C01780=1012.126,212.410,-136.881,-33.428,76.064,-33.422
C01781=1012.128,212.654,-136.908,-33.436,76.075,-33.431
C01782=1012.129,212.897,-136.935,-33.444,76.085,-33.440
C01783=1012.131,213.142,-136.961,-33.452,76.095,-33.450
C01784=1012.133,213.385,-136.987,-33.459,76.106,-33.457
C01785=1012.135,213.629,-137.015,-33.468,76.116,-33.467
C01786=1012.138,213.873,-137.042,-33.476,76.127,-33.476
C01787=1012.140,214.117,-137.068,-33.485,76.137,-33.487
C01788=1012.142,214.361,-137.095,-33.493,76.147,-33.496
C01789=1012.144,214.607,-137.122,-33.501,76.158,-33.504
C01790=1012.146,214.852,-137.149,-33.509,76.168,-33.515
C01791=1012.149,215.097,-137.177,-33.518,76.179,-33.524
C01792=1012.151,215.342,-137.204,-33.526,76.189,-33.534
C01793=1012.152,215.587,-137.231,-33.534,76.200,-33.543
C01794=1012.155,215.832,-137.258,-33.543,76.210,-33.554
C01795=1012.157,216.079,-137.285,-33.552,76.221,-33.563
C01796=1012.160,216.324,-137.312,-33.561,76.231,-33.574
C01797=1012.161,216.570,-137.339,-33.569,76.242,-33.583
C01798=1012.164,216.818,-137.366,-33.577,76.253,-33.592
C01799=1012.167,217.073,-137.394,-33.584,76.263,-33.599
C01800=1012.169,217.333,-137.423,-33.593,76.274,-33.610
C01801=1012.171,217.597,-137.452,-33.601,76.285,-33.619
C01802=1012.174,217.878,-137.484,-33.611,76.297,-33.630
C01803=1012.176,218.167,-137.515,-33.622,76.309,-33.643
C01804=1012.179,218.460,-137.547,-33.633,76.322,-33.656
C01805=1012.182,218.757,-137.580,-33.644,76.334,-33.669
C01806=1012.185,219.060,-137.614,-33.655,76.346,-33.682
C01807=1012.187,219.356,-137.647,-33.666,76.358,-33.695
C01808=1012.190,219.638,-137.678,-33.676,76.370,-33.706
C01809=1012.193,219.909,-137.708,-33.686,76.382,-33.717
C01810=1012.195,220.170,-137.737,-33.693,76.393,-33.725
C01811=1012.197,220.419,-137.765,-33.702,76.404,-33.734
C01812=1012.200,220.665,-137.792,-33.709,76.414,-33.743
C01813=1012.202,220.911,-137.819,-33.718,76.424,-33.752
C01814=1012.205,221.156,-137.846,-33.727,76.434,-33.763
C01815=1012.208,221.402,-137.874,-33.736,76.444,-33.774
C01816=1012.210,221.648,-137.901,-33.743,76.454,-33.782
C01817=1012.211,221.894,-137.929,-33.753,76.464,-33.793
C01818=1012.214,222.140,-137.956,-33.761,76.474,-33.802
C01819=1012.216,222.385,-137.983,-33.769,76.483,-33.811
C01820=1012.219,222.630,-138.011,-33.778,76.493,-33.822
C01821=1012.222,222.876,-138.038,-33.785,76.503,-33.829
C01822=1012.224,223.122,-138.065,-33.794,76.513,-33.840
C01823=1012.227,223.368,-138.093,-33.803,76.524,-33.850
C01824=1012.229,223.614,-138.120,-33.812,76.534,-33.861
C01825=1012.231,223.859,-138.147,-33.822,76.545,-33.873
C01826=1012.234,224.105,-138.175,-33.831,76.556,-33.882
C01827=1012.236,224.351,-138.203,-33.840,76.566,-33.893
C01828=1012.238,224.597,-138.230,-33.849,76.575,-33.902
C01829=1012.241,224.842,-138.258,-33.857,76.585,-33.912
C01830=1012.243,225.088,-138.285,-33.864,76.595,-33.919
C01831=1012.246,225.334,-138.313,-33.873,76.605,-33.930
C01832=1012.248,225.579,-138.340,-33.883,76.615,-33.942
C01833=1012.251,225.825,-138.367,-33.890,76.625,-33.949
C01834=1012.253,226.071,-138.394,-33.900,76.635,-33.961
C01835=1012.256,226.316,-138.423,-33.908,76.646,-33.970
C01836=1012.258,226.562,-138.450,-33.918,76.656,-33.982
C01837=1012.261,226.807,-138.477,-33.928,76.667,-33.993
C01838=1012.264,227.053,-138.505,-33.937,76.677,-34.003
C01839=1012.266,227.299,-138.532,-33.945,76.686,-34.012
C01840=1012.268,227.545,-138.560,-33.953,76.695,-34.021
C01841=1012.271,227.790,-138.588,-33.962,76.706,-34.031
C01842=1012.273,228.036,-138.615,-33.970,76.715,-34.041
C01843=1012.276,228.282,-138.642,-33.980,76.725,-34.052
C01844=1012.279,228.527,-138.671,-33.990,76.735,-34.064
C01845=1012.281,228.773,-138.698,-33.998,76.746,-34.073
C01846=1012.284,229.018,-138.726,-34.007,76.757,-34.083
C01847=1012.286,229.264,-138.753,-34.017,76.767,-34.095
C01848=1012.289,229.510,-138.780,-34.026,76.777,-34.105
C01849=1012.291,229.755,-138.808,-34.034,76.787,-34.114
C01850=1012.294,230.001,-138.836,-34.043,76.796,-34.124
C01851=1012.297,230.246,-138.863,-34.051,76.805,-34.133
C01852=1012.300,230.492,-138.891,-34.061,76.815,-34.145
C01853=1012.301,230.738,-138.919,-34.069,76.824,-34.154
C01854=1012.304,230.984,-138.947,-34.079,76.834,-34.166
C01855=1012.307,231.229,-138.974,-34.087,76.844,-34.174
C01856=1012.310,231.475,-139.002,-34.097,76.854,-34.186
C01857=1012.313,231.721,-139.030,-34.106,76.865,-34.196
C01858=1012.315,231.966,-139.057,-34.116,76.875,-34.208
C01859=1012.318,232.212,-139.085,-34.125,76.886,-34.218
C01860=1012.320,232.457,-139.113,-34.134,76.895,-34.227
C01861=1012.323,232.703,-139.141,-34.142,76.904,-34.237
C01862=1012.326,232.948,-139.168,-34.152,76.913,-34.248
C01863=1012.329,233.193,-139.197,-34.161,76.924,-34.259
C01864=1012.332,233.439,-139.224,-34.169,76.933,-34.268
C01865=1012.334,233.684,-139.252,-34.179,76.943,-34.280
C01866=1012.337,233.931,-139.279,-34.188,76.952,-34.290
C01867=1012.340,234.175,-139.307,-34.197,76.963,-34.300
C01868=1012.342,234.421,-139.336,-34.207,76.973,-34.312
C01869=1012.345,234.668,-139.363,-34.217,76.983,-34.322
C01870=1012.347,234.912,-139.391,-34.227,76.993,-34.334
C01871=1012.350,235.158,-139.419,-34.236,77.003,-34.344
C01872=1012.353,235.404,-139.447,-34.244,77.012,-34.354
C01873=1012.356,235.649,-139.475,-34.253,77.021,-34.364
C01874=1012.359,235.895,-139.503,-34.262,77.030,-34.374
C01875=1012.361,236.140,-139.531,-34.270,77.039,-34.384
C01876=1012.364,236.385,-139.559,-34.281,77.049,-34.396
C01877=1012.368,236.631,-139.587,-34.290,77.060,-34.406
C01878=1012.370,236.876,-139.614,-34.299,77.069,-34.416
C01879=1012.373,237.122,-139.642,-34.308,77.080,-34.426
C01880=1012.376,237.368,-139.670,-34.320,77.091,-34.441
C01881=1012.378,237.612,-139.698,-34.328,77.099,-34.449
C01882=1012.382,237.858,-139.726,-34.336,77.109,-34.459
C01883=1012.385,238.104,-139.754,-34.345,77.118,-34.469
C01884=1012.387,238.350,-139.782,-34.355,77.126,-34.481
C01885=1012.389,238.595,-139.810,-34.364,77.135,-34.491
C01886=1012.392,238.841,-139.838,-34.373,77.146,-34.501
C01887=1012.396,239.086,-139.867,-34.382,77.155,-34.511
C01888=1012.398,239.331,-139.894,-34.393,77.165,-34.524
C01889=1012.401,239.577,-139.923,-34.403,77.176,-34.534
C01890=1012.404,239.822,-139.951,-34.413,77.186,-34.546
C01891=1012.407,240.067,-139.979,-34.423,77.197,-34.557
C01892=1012.410,240.313,-140.007,-34.431,77.204,-34.567
C01893=1012.413,240.558,-140.035,-34.440,77.213,-34.577
C01894=1012.416,240.804,-140.063,-34.449,77.223,-34.587
C01895=1012.419,241.050,-140.091,-34.458,77.232,-34.598
C01896=1012.422,241.295,-140.119,-34.467,77.241,-34.608
C01897=1012.425,241.540,-140.147,-34.478,77.251,-34.620
C01898=1012.428,241.786,-140.175,-34.487,77.260,-34.631
C01899=1012.431,242.031,-140.204,-34.498,77.270,-34.643
C01900=1012.434,242.276,-140.231,-34.507,77.281,-34.654
C01901=1012.436,242.522,-140.260,-34.518,77.291,-34.666
C01902=1012.439,242.768,-140.288,-34.526,77.301,-34.675
C01903=1012.443,243.013,-140.317,-34.536,77.309,-34.687
C01904=1012.446,243.258,-140.345,-34.544,77.318,-34.695
C01905=1012.448,243.503,-140.373,-34.554,77.326,-34.708
C01906=1012.451,243.749,-140.401,-34.563,77.335,-34.718
C01907=1012.454,243.994,-140.429,-34.573,77.344,-34.728
C01908=1012.457,244.240,-140.458,-34.583,77.354,-34.741
C01909=1012.461,244.485,-140.486,-34.592,77.364,-34.750
C01910=1012.464,244.731,-140.515,-34.603,77.374,-34.762
C01911=1012.467,244.975,-140.542,-34.614,77.384,-34.775
C01912=1012.470,245.221,-140.571,-34.624,77.395,-34.786
C01913=1012.473,245.466,-140.600,-34.633,77.404,-34.797
C01914=1012.476,245.712,-140.628,-34.641,77.412,-34.807
C01915=1012.479,245.957,-140.656,-34.651,77.421,-34.817
C01916=1012.482,246.203,-140.685,-34.659,77.429,-34.826
C01917=1012.485,246.448,-140.714,-34.668,77.438,-34.836
C01918=1012.488,246.694,-140.742,-34.678,77.447,-34.849
C01919=1012.491,246.939,-140.769,-34.688,77.457,-34.860
C01920=1012.494,247.184,-140.798,-34.698,77.467,-34.871
C01921=1012.497,247.429,-140.827,-34.709,77.477,-34.884
C01922=1012.500,247.675,-140.855,-34.719,77.487,-34.895
C01923=1012.504,247.920,-140.884,-34.730,77.497,-34.908
C01924=1012.507,248.165,-140.912,-34.738,77.506,-34.916
C01925=1012.510,248.410,-140.941,-34.749,77.514,-34.929
C01926=1012.513,248.656,-140.969,-34.756,77.522,-34.937
C01927=1012.517,248.901,-140.998,-34.767,77.531,-34.950
C01928=1012.520,249.147,-141.026,-34.776,77.540,-34.961
C01929=1012.523,249.391,-141.055,-34.786,77.549,-34.971
C01930=1012.526,249.637,-141.083,-34.796,77.558,-34.982
C01931=1012.529,249.883,-141.112,-34.807,77.568,-34.995
C01932=1012.532,250.128,-141.141,-34.817,77.579,-35.007
C01933=1012.535,250.374,-141.169,-34.827,77.588,-35.017
C01934=1012.539,250.619,-141.198,-34.838,77.598,-35.031
C01935=1012.542,250.864,-141.226,-34.846,77.606,-35.039
C01936=1012.545,251.109,-141.255,-34.857,77.615,-35.052
C01937=1012.549,251.354,-141.284,-34.865,77.623,-35.061
C01938=1012.552,251.600,-141.312,-34.875,77.631,-35.073
C01939=1012.555,251.845,-141.341,-34.885,77.640,-35.084
C01940=1012.559,252.090,-141.369,-34.895,77.650,-35.095
C01941=1012.562,252.335,-141.398,-34.905,77.659,-35.106
C01942=1012.565,252.580,-141.427,-34.916,77.669,-35.120
C01943=1012.568,252.826,-141.455,-34.925,77.679,-35.129
C01944=1012.571,253.071,-141.484,-34.937,77.689,-35.142
C01945=1012.575,253.316,-141.513,-34.946,77.698,-35.153
C01946=1012.578,253.562,-141.541,-34.956,77.705,-35.164
C01947=1012.581,253.807,-141.570,-34.965,77.714,-35.175
C01948=1012.584,254.052,-141.599,-34.974,77.722,-35.186
C01949=1012.588,254.297,-141.628,-34.984,77.731,-35.197
C01950=1012.591,254.542,-141.656,-34.994,77.740,-35.208
C01951=1012.594,254.787,-141.685,-35.004,77.749,-35.219
C01952=1012.598,255.032,-141.714,-35.014,77.759,-35.231
C01953=1012.602,255.278,-141.743,-35.026,77.768,-35.244
C01954=1012.605,255.523,-141.773,-35.036,77.778,-35.255
C01955=1012.608,255.769,-141.801,-35.047,77.788,-35.267
C01956=1012.611,256.014,-141.830,-35.058,77.797,-35.280
C01957=1012.615,256.259,-141.858,-35.066,77.805,-35.289
C01958=1012.618,256.504,-141.887,-35.075,77.813,-35.300
C01959=1012.621,256.749,-141.916,-35.085,77.822,-35.311
C01960=1012.625,256.994,-141.945,-35.095,77.829,-35.322
C01961=1012.629,257.239,-141.974,-35.105,77.838,-35.334
C01962=1012.632,257.484,-142.003,-35.115,77.848,-35.345
C01963=1012.635,257.730,-142.031,-35.125,77.857,-35.356
C01964=1012.638,257.975,-142.061,-35.137,77.867,-35.370
C01965=1012.641,258.220,-142.090,-35.149,77.876,-35.384
C01966=1012.645,258.466,-142.119,-35.158,77.886,-35.393
C01967=1012.659,259.701,-142.272,-34.356,78.117,-34.079
C01968=1012.662,260.109,-142.326,-34.065,78.179,-33.616
C01969=1012.663,260.518,-142.380,-33.799,78.275,-33.178
C01970=1012.664,260.926,-142.437,-33.509,78.350,-32.716
C01971=1012.663,261.334,-142.494,-33.211,78.423,-32.244
C01972=1012.662,261.743,-142.552,-32.937,78.531,-31.799
C01973=1012.659,262.151,-142.613,-32.628,78.602,-31.316
C01974=1012.656,262.559,-142.674,-32.326,78.691,-30.842
C01975=1012.652,262.968,-142.738,-32.000,78.752,-30.341
C01976=1012.647,263.375,-142.801,-31.691,78.850,-29.859
C01977=1012.641,263.782,-142.869,-31.353,78.913,-29.346
C01978=1012.634,264.190,-142.936,-31.022,78.991,-28.841
C01979=1012.626,264.598,-143.004,-30.698,79.097,-28.344
C01980=1012.617,265.005,-143.076,-30.337,79.150,-27.807
C01981=1012.607,265.413,-143.146,-29.992,79.240,-27.288
C01982=1012.595,265.819,-143.219,-29.639,79.333,-26.761
C01983=1012.583,266.227,-143.293,-29.273,79.414,-26.220
C01984=1012.570,266.634,-143.369,-28.897,79.484,-25.668
C01985=1012.557,267.041,-143.447,-28.513,79.562,-25.107
C01986=1012.542,267.447,-143.526,-28.130,79.653,-24.550
C01987=1012.526,267.853,-143.606,-27.726,79.712,-23.968
C01988=1012.509,268.259,-143.688,-27.327,79.807,-23.393
C01989=1012.491,268.665,-143.771,-26.911,79.882,-22.800
C01990=1012.472,269.072,-143.856,-26.488,79.952,-22.199
C01991=1012.452,269.478,-143.941,-26.063,80.058,-21.600
C01992=1012.431,269.883,-144.028,-25.620,80.129,-20.978
C01993=1012.409,270.288,-144.117,-25.170,80.220,-20.351
C01994=1012.386,270.694,-144.209,-24.709,80.277,-19.709
C01995=1012.361,271.098,-144.300,-24.242,80.371,-19.066
C01996=1012.337,271.504,-144.394,-23.762,80.439,-18.406
C01997=1012.311,271.908,-144.488,-23.272,80.520,-17.736
C01998=1012.284,272.313,-144.584,-22.768,80.606,-17.054
C01999=1012.255,272.717,-144.682,-22.257,80.673,-16.361
C02000=1012.227,273.121,-144.780,-21.728,80.775,-15.656
C02001=1012.197,273.526,-144.881,-21.193,80.845,-14.939
C02002=1012.165,273.929,-144.984,-20.642,80.918,-14.206
C02003=1012.133,274.333,-145.088,-20.080,80.993,-13.462
C02004=1012.099,274.736,-145.192,-19.496,81.082,-12.698
C02005=1012.065,275.140,-145.300,-18.902,81.160,-11.919
C02006=1012.030,275.542,-145.408,-18.296,81.231,-11.129
C02007=1011.993,275.945,-145.518,-17.671,81.309,-10.319
C02008=1011.955,276.347,-145.629,-17.029,81.388,-9.493
C02009=1011.916,276.749,-145.742,-16.370,81.468,-8.648
C02010=1011.877,277.150,-145.857,-15.699,81.540,-7.791
C02011=1011.836,277.552,-145.972,-14.999,81.625,-6.906
C02012=1011.794,277.954,-146.091,-14.306,81.682,-6.021
///RCONF 0,0,0,0,0,0,0,0,0,0,0,0,0,0,0,0,0,0,0,0,0,0,0,0
C02013=1011.751,278.355,-146.209,-13.561,81.772,-5.092
C02014=1011.707,278.755,-146.330,-12.812,81.847,-4.154
C02015=1011.662,279.156,-146.453,-12.063,81.908,-3.213
C02016=1011.615,279.556,-146.576,-11.266,81.987,-2.228
C02017=1011.568,279.956,-146.702,-10.466,82.055,-1.236
C02018=1011.520,280.355,-146.828,-9.621,82.131,-0.200
C02019=1011.469,280.754,-146.957,-8.748,82.208,0.865
C02020=1011.418,281.153,-147.087,-7.854,82.282,1.952
C02021=1011.366,281.551,-147.219,-6.951,82.345,3.054
C02022=1011.313,281.949,-147.352,-5.979,82.425,4.221
C02023=1011.286,282.148,-147.420,-5.489,82.462,4.808
C02024=1011.258,282.347,-147.487,-5.001,82.493,5.398
C02025=1011.231,282.546,-147.556,-4.501,82.528,5.997
C02026=1011.202,282.744,-147.624,-3.990,82.563,6.608
C02027=1011.174,282.943,-147.693,-3.493,82.589,7.207
C02028=1011.145,283.140,-147.763,-2.965,82.625,7.834
C02029=1011.117,283.339,-147.832,-2.417,82.663,8.482
C02030=1011.088,283.536,-147.903,-1.899,82.688,9.103
C02031=1011.058,283.735,-147.974,-1.341,82.723,9.762
C02032=1011.028,283.933,-148.044,-0.760,82.763,10.442
C02033=1010.998,284.131,-148.116,-0.205,82.791,11.101
C02034=1010.968,284.328,-148.188,0.380,82.825,11.786
C02035=1010.937,284.526,-148.261,0.936,82.848,12.448
C02036=1010.906,284.724,-148.333,1.533,82.881,13.146
C02037=1010.875,284.921,-148.407,2.133,82.910,13.849
C02038=1010.843,285.118,-148.481,2.711,82.931,14.533
C02039=1010.811,285.314,-148.556,3.329,82.960,15.256
C02040=1010.779,285.512,-148.629,3.994,82.998,16.021
C02041=1010.746,285.709,-148.704,4.634,83.026,16.764
C02042=1010.713,285.905,-148.781,5.281,83.054,17.515
C02043=1010.681,286.101,-148.856,5.929,83.078,18.270
C02044=1010.646,286.298,-148.933,6.600,83.104,19.047
C02045=1010.612,286.494,-149.010,7.280,83.130,19.833
C02046=1010.579,286.690,-149.088,7.927,83.145,20.590
C02047=1010.544,286.886,-149.166,8.623,83.169,21.393
C02048=1010.508,287.083,-149.243,9.382,83.202,22.256
C02049=1010.474,287.278,-149.322,10.083,83.219,23.067
C02050=1010.438,287.473,-149.402,10.786,83.235,23.882
C02051=1010.403,287.669,-149.481,11.547,83.260,24.750
C02052=1010.366,287.864,-149.560,12.362,83.290,25.670
C02053=1010.329,288.059,-149.642,13.098,83.304,26.518
C02054=1010.292,288.254,-149.722,13.896,83.326,27.424
C02055=1010.256,288.449,-149.804,14.648,83.337,28.290
C02056=1010.218,288.644,-149.886,15.421,83.350,29.176
C02057=1010.179,288.838,-149.968,16.267,83.370,30.130
C02058=1010.141,289.032,-150.051,17.100,83.386,31.073
C02059=1010.103,289.226,-150.135,17.936,83.400,32.020
C02060=1010.064,289.420,-150.218,18.754,83.409,32.953
C02061=1010.025,289.614,-150.303,19.617,83.421,33.928
C02062=1009.985,289.808,-150.388,20.451,83.428,34.877
C02063=1009.945,290.001,-150.473,21.322,83.435,35.864
C02064=1009.905,290.195,-150.559,22.218,83.443,36.873
C02065=1009.863,290.387,-150.646,23.058,83.443,37.831
C02066=1009.822,290.580,-150.733,23.981,83.450,38.868
C02067=1009.781,290.773,-150.820,24.882,83.451,39.885
C02068=1009.739,290.965,-150.908,25.775,83.449,40.896
C02069=1009.697,291.158,-150.996,26.753,83.453,41.989
C02070=1009.654,291.350,-151.085,27.660,83.449,43.015
C02071=1009.611,291.542,-151.174,28.628,83.446,44.100
C02072=1009.568,291.733,-151.265,29.517,83.435,45.111
C02073=1009.525,291.925,-151.356,30.507,83.430,46.219
C02074=1009.480,292.117,-151.446,31.413,83.416,47.248
C02075=1009.436,292.307,-151.539,32.334,83.401,48.291
C02076=1009.391,292.498,-151.630,33.357,83.392,49.433
C02077=1009.346,292.689,-151.723,34.361,83.379,50.555
C02078=1009.300,292.879,-151.815,35.346,83.362,51.662
C02079=1009.254,293.069,-151.910,36.301,83.341,52.740
C02080=1009.208,293.259,-152.004,37.296,83.320,53.859
C02081=1009.161,293.449,-152.098,38.275,83.295,54.962
C02082=1009.114,293.639,-152.194,39.247,83.269,56.059
C02083=1009.066,293.828,-152.290,40.282,83.243,57.217
C02084=1009.018,294.017,-152.386,41.233,83.210,58.296
C02085=1008.970,294.205,-152.483,42.268,83.181,59.453
C02086=1008.921,294.394,-152.581,43.222,83.144,60.537
C02087=1008.871,294.582,-152.679,44.231,83.108,61.672
C02088=1008.822,294.770,-152.778,45.232,83.070,62.798
C02089=1008.772,294.958,-152.876,46.245,83.029,63.938
C02090=1008.721,295.145,-152.977,47.183,82.983,65.008
C02091=1008.670,295.333,-153.077,48.203,82.938,66.154
C02092=1008.619,295.519,-153.179,49.113,82.886,67.199
C02093=1008.567,295.707,-153.281,50.086,82.835,68.300
C02094=1008.515,295.893,-153.382,51.138,82.786,69.476
C02095=1008.462,296.079,-153.485,52.083,82.728,70.554
C02096=1008.409,296.265,-153.588,53.034,82.670,71.635
C02097=1008.356,296.451,-153.692,53.992,82.610,72.725
C02098=1008.302,296.635,-153.798,54.922,82.546,73.787
C02099=1008.247,296.821,-153.903,55.868,82.480,74.865
C02100=1008.193,297.006,-154.009,56.789,82.411,75.920
C02101=1008.138,297.189,-154.115,57.702,82.340,76.967
C02102=1008.082,297.374,-154.222,58.657,82.268,78.053
C02103=1008.025,297.557,-154.330,59.493,82.190,79.028
C02104=1007.969,297.741,-154.438,60.423,82.113,80.089
C02105=1007.912,297.925,-154.547,61.329,82.032,81.129
C02106=1007.855,298.107,-154.657,62.166,81.948,82.104
C02107=1007.797,298.289,-154.767,63.085,81.864,83.153
C02108=1007.738,298.471,-154.878,63.950,81.776,84.153
C02109=1007.679,298.653,-154.989,64.822,81.686,85.159
C02110=1007.620,298.835,-155.101,65.608,81.592,86.085
C02111=1007.559,299.016,-155.214,66.450,81.496,87.062
C02112=1007.499,299.196,-155.327,67.303,81.399,88.048
C02113=1007.439,299.377,-155.440,68.132,81.299,89.011
C02114=1007.377,299.558,-155.556,68.904,81.195,89.923
C02115=1007.315,299.737,-155.671,69.683,81.090,90.839
C02116=1007.253,299.917,-155.786,70.456,80.982,91.748
C02117=1007.190,300.095,-155.903,71.208,80.872,92.639
C02118=1007.128,300.274,-156.021,71.962,80.760,93.530
C02119=1007.064,300.452,-156.139,72.695,80.645,94.402
C02120=1006.999,300.630,-156.257,73.408,80.527,95.254
C02121=1006.934,300.807,-156.376,74.180,80.408,96.158
C02122=1006.870,300.984,-156.496,74.851,80.286,96.971
C02123=1006.804,301.161,-156.617,75.585,80.161,97.838
C02124=1006.738,301.337,-156.738,76.228,80.036,98.624
C02125=1006.671,301.513,-156.860,76.950,79.906,99.478
C02126=1006.604,301.689,-156.983,77.596,79.776,100.264
C02127=1006.536,301.863,-157.106,78.232,79.642,101.040
C02128=1006.468,302.038,-157.230,78.893,79.506,101.838
C02129=1006.399,302.212,-157.355,79.481,79.369,102.570
C02130=1006.330,302.387,-157.480,80.107,79.229,103.332
C02131=1006.260,302.559,-157.606,80.749,79.087,104.107
C02132=1006.190,302.733,-157.733,81.359,78.943,104.854
C02133=1006.120,302.905,-157.860,81.925,78.797,105.560
C02134=1006.048,303.076,-157.988,82.506,78.649,106.278
C02135=1005.976,303.247,-158.117,83.069,78.499,106.979
C02136=1005.904,303.418,-158.246,83.618,78.347,107.667
C02137=1005.832,303.589,-158.376,84.164,78.194,108.349
C02138=1005.758,303.759,-158.507,84.697,78.038,109.019
C02139=1005.684,303.929,-158.639,85.209,77.880,109.672
C02140=1005.610,304.098,-158.770,85.770,77.719,110.361
C02141=1005.535,304.267,-158.904,86.250,77.559,110.982
C02142=1005.460,304.434,-159.037,86.784,77.394,111.645
C02143=1005.384,304.602,-159.172,87.243,77.229,112.247
C02144=1005.307,304.769,-159.306,87.757,77.061,112.890
C02145=1005.231,304.935,-159.443,88.224,76.892,113.494
C02146=1005.152,305.101,-159.579,88.679,76.722,114.086
C02147=1005.075,305.267,-159.715,89.148,76.549,114.686
C02148=1004.996,305.431,-159.854,89.565,76.377,115.243
C02149=1004.917,305.596,-159.992,90.008,76.201,115.819
C02150=1004.837,305.759,-160.131,90.470,76.023,116.407
C02151=1004.758,305.923,-160.271,90.900,75.845,116.967
C02152=1004.677,306.086,-160.412,91.302,75.666,117.503
C02153=1004.595,306.247,-160.552,91.711,75.484,118.043
C02154=1004.513,306.409,-160.694,92.113,75.301,118.576
C02155=1004.432,306.570,-160.837,92.500,75.118,119.093
C02156=1004.349,306.730,-160.981,92.888,74.932,119.611
C02157=1004.265,306.889,-161.125,93.267,74.745,120.119
C02158=1004.182,307.049,-161.270,93.628,74.557,120.612
C02159=1004.098,307.207,-161.414,94.031,74.366,121.133
C02160=1004.013,307.365,-161.561,94.357,74.177,121.596
C02161=1003.928,307.523,-161.707,94.734,73.983,122.093
C02162=1003.842,307.679,-161.854,95.069,73.790,122.558
C02163=1003.755,307.835,-162.002,95.414,73.595,123.028
C02164=1003.668,307.990,-162.150,95.770,73.398,123.502
C02165=1003.581,308.145,-162.300,96.104,73.201,123.959
C02166=1003.493,308.299,-162.451,96.409,73.005,124.391
C02167=1003.404,308.452,-162.601,96.737,72.806,124.839
C02168=1003.315,308.605,-162.752,97.028,72.608,125.256
C02169=1003.225,308.757,-162.904,97.324,72.409,125.675
C02170=1003.136,308.909,-163.056,97.664,72.207,126.122
C02171=1002.979,309.171,-163.323,98.183,71.856,126.844
C02172=1002.819,309.430,-163.591,98.681,71.503,127.543
C02173=1003.018,309.121,-163.890,77.094,71.863,112.900
C02174=1003.161,308.887,-163.649,76.172,72.173,111.744
C02175=1003.302,308.651,-163.409,75.210,72.476,110.550
C02176=1003.392,308.501,-163.258,74.548,72.665,109.749
C02177=1003.481,308.350,-163.107,73.924,72.852,108.972
C02178=1003.569,308.198,-162.955,73.303,73.038,108.192
C02179=1003.657,308.046,-162.806,72.631,73.220,107.370
C02180=1003.745,307.893,-162.657,71.982,73.400,106.562
C02181=1003.831,307.739,-162.508,71.294,73.578,105.719
C02182=1003.918,307.585,-162.361,70.582,73.751,104.857
C02183=1004.004,307.429,-162.214,69.873,73.922,103.991
C02184=1004.090,307.274,-162.067,69.167,74.092,103.123
C02185=1004.174,307.117,-161.922,68.410,74.257,102.212
C02186=1004.258,306.960,-161.776,67.703,74.421,101.336
C02187=1004.342,306.802,-161.632,66.915,74.579,100.395
C02188=1004.425,306.645,-161.488,66.163,74.735,99.479
C02189=1004.508,306.485,-161.345,65.388,74.887,98.543
C02190=1004.590,306.327,-161.203,64.598,75.036,97.590
C02191=1004.672,306.167,-161.061,63.808,75.181,96.636
C02192=1004.753,306.006,-160.920,62.999,75.324,95.661
C02193=1004.834,305.845,-160.780,62.174,75.462,94.673
C02194=1004.914,305.683,-160.639,61.357,75.598,93.687
C02195=1004.993,305.521,-160.501,60.507,75.728,92.674
C02196=1005.073,305.358,-160.362,59.625,75.854,91.630
C02197=1005.151,305.195,-160.226,58.758,75.978,90.598
C02198=1005.229,305.031,-160.088,57.910,76.100,89.575
C02199=1005.307,304.866,-159.952,57.018,76.215,88.518
C02200=1005.384,304.701,-159.816,56.131,76.328,87.459
C02201=1005.460,304.535,-159.681,55.236,76.438,86.393
C02202=1005.536,304.370,-159.548,54.297,76.540,85.291
C02203=1005.611,304.203,-159.413,53.405,76.643,84.223
C02204=1005.687,304.036,-159.281,52.450,76.737,83.103
C02205=1005.761,303.868,-159.148,51.546,76.831,82.024
C02206=1005.835,303.700,-159.018,50.569,76.917,80.883
C02207=1005.908,303.532,-158.886,49.640,77.002,79.780
C02208=1005.981,303.363,-158.757,48.693,77.083,78.660
C02209=1006.053,303.193,-158.628,47.738,77.159,77.534
C02210=1006.125,303.024,-158.498,46.789,77.233,76.412
C02211=1006.196,302.853,-158.371,45.831,77.301,75.282
C02212=1006.267,302.682,-158.244,44.865,77.365,74.144
C02213=1006.338,302.511,-158.116,43.918,77.428,73.021
C02214=1006.407,302.339,-157.990,42.937,77.484,71.868
C02215=1006.477,302.166,-157.865,41.940,77.534,70.703
C02216=1006.545,301.994,-157.741,40.968,77.582,69.560
C02217=1006.613,301.821,-157.616,40.027,77.631,68.439
C02218=1006.681,301.647,-157.494,39.047,77.670,67.289
C02219=1006.748,301.473,-157.370,38.094,77.710,66.162
C02220=1006.815,301.298,-157.249,37.138,77.745,65.030
C02221=1006.882,301.123,-157.128,36.143,77.771,63.867
C02222=1006.947,300.948,-157.006,35.217,77.802,62.764
C02223=1007.013,300.773,-156.887,34.240,77.821,61.619
C02224=1007.077,300.597,-156.768,33.314,77.844,60.517
C02225=1007.142,300.420,-156.650,32.341,77.856,59.376
C02226=1007.205,300.244,-156.531,31.418,77.871,58.279
C02227=1007.269,300.066,-156.414,30.495,77.882,57.183
C02228=1007.332,299.888,-156.297,29.571,77.888,56.088
C02229=1007.394,299.710,-156.181,28.661,77.893,55.005
C02230=1007.456,299.532,-156.066,27.756,77.894,53.928
C02231=1007.517,299.353,-155.951,26.858,77.892,52.859
C02232=1007.578,299.174,-155.837,25.983,77.890,51.811
C02233=1007.638,298.994,-155.723,25.092,77.881,50.750
C02234=1007.698,298.815,-155.611,24.204,77.867,49.695
C02235=1007.758,298.634,-155.499,23.334,77.853,48.656
C02236=1007.817,298.454,-155.387,22.510,77.843,47.658
C02237=1007.875,298.273,-155.277,21.655,77.822,46.636
C02238=1007.934,298.091,-155.166,20.824,77.802,45.636
C02239=1007.992,297.910,-155.058,19.979,77.774,44.626
C02240=1008.048,297.728,-154.948,19.193,77.754,43.669
C02241=1008.105,297.546,-154.840,18.390,77.726,42.700
C02242=1008.162,297.363,-154.732,17.590,77.694,41.735
C02243=1008.217,297.181,-154.625,16.842,77.671,40.814
C02244=1008.272,296.998,-154.519,16.062,77.635,39.871
C02245=1008.327,296.813,-154.413,15.317,77.602,38.959
C02246=1008.382,296.631,-154.307,14.584,77.569,38.059
C02247=1008.436,296.446,-154.203,13.851,77.530,37.162
C02248=1008.489,296.262,-154.098,13.140,77.493,36.285
C02249=1008.543,296.078,-153.995,12.431,77.453,35.412
C02250=1008.596,295.892,-153.892,11.735,77.411,34.552
C02251=1008.648,295.707,-153.789,11.063,77.371,33.716
C02252=1008.700,295.522,-153.688,10.360,77.317,32.856
C02253=1008.751,295.335,-153.587,9.699,77.272,32.032
C02254=1008.803,295.150,-153.486,9.077,77.233,31.245
C02255=1008.853,294.964,-153.386,8.421,77.180,30.431
C02256=1008.903,294.776,-153.286,7.813,77.138,29.660
C02257=1008.953,294.590,-153.188,7.191,77.086,28.880
C02258=1009.002,294.402,-153.090,6.576,77.033,28.107
C02259=1009.052,294.215,-152.992,5.976,76.979,27.351
C02260=1009.100,294.027,-152.894,5.406,76.932,26.619
C02261=1009.148,293.839,-152.798,4.814,76.872,25.874
C02262=1009.196,293.652,-152.702,4.267,76.824,25.168
C02263=1009.243,293.463,-152.607,3.703,76.765,24.451
C02264=1009.290,293.275,-152.512,3.160,76.711,23.751
C02265=1009.337,293.086,-152.417,2.630,76.658,23.067
C02266=1009.383,292.897,-152.323,2.104,76.600,22.388
C02267=1009.429,292.707,-152.230,1.595,76.546,21.724
C02268=1009.474,292.518,-152.138,1.089,76.488,21.065
C02269=1009.519,292.328,-152.046,0.585,76.427,20.412
C02270=1009.564,292.137,-151.954,0.085,76.362,19.765
C02271=1009.608,291.948,-151.863,-0.381,76.309,19.146
C02272=1009.651,291.757,-151.772,-0.839,76.256,18.537
C02273=1009.695,291.567,-151.682,-1.306,76.194,17.923
C02274=1009.739,291.376,-151.592,-1.745,76.141,17.332
C02275=1009.782,291.185,-151.503,-2.198,76.078,16.733
C02276=1009.823,290.993,-151.415,-2.627,76.022,16.156
C02277=1009.866,290.802,-151.327,-3.071,75.954,15.568
C02278=1009.907,290.611,-151.239,-3.488,75.897,15.005
C02279=1009.948,290.419,-151.152,-3.897,75.839,14.450
C02280=1009.990,290.226,-151.066,-4.311,75.774,13.893
C02281=1010.030,290.034,-150.980,-4.699,75.721,13.358
C02282=1010.071,289.842,-150.894,-5.094,75.657,12.822
C02283=1010.110,289.649,-150.808,-5.476,75.598,12.298
C02284=1010.149,289.456,-150.724,-5.851,75.541,11.780
C02285=1010.189,289.263,-150.640,-6.226,75.478,11.264
C02286=1010.227,289.070,-150.557,-6.583,75.421,10.767
C02287=1010.266,288.877,-150.474,-6.943,75.360,10.266
C02288=1010.305,288.683,-150.391,-7.301,75.296,9.771
C02289=1010.341,288.489,-150.309,-7.655,75.230,9.280
C02290=1010.379,288.296,-150.227,-7.991,75.173,8.805
C02291=1010.416,288.101,-150.146,-8.317,75.120,8.339
C02292=1010.453,287.907,-150.066,-8.650,75.056,7.870
C02293=1010.489,287.713,-149.985,-8.967,75.003,7.415
C02294=1010.526,287.518,-149.906,-9.300,74.931,6.949
C02295=1010.561,287.324,-149.826,-9.618,74.867,6.498
C02296=1010.596,287.129,-149.748,-9.919,74.814,6.059
C02297=1010.632,286.934,-149.668,-10.214,74.761,5.627
C02298=1010.666,286.739,-149.591,-10.525,74.691,5.185
C02299=1010.701,286.544,-149.514,-10.816,74.633,4.763
C02300=1010.735,286.349,-149.436,-11.094,74.584,4.348
C02301=1010.768,286.153,-149.360,-11.376,74.526,3.934
C02302=1010.801,285.957,-149.283,-11.655,74.467,3.523
C02303=1010.834,285.761,-149.208,-11.927,74.413,3.120
C02304=1010.867,285.566,-149.132,-12.198,74.353,2.719
C02305=1010.900,285.369,-149.057,-12.462,74.296,2.326
C02306=1010.932,285.173,-148.984,-12.733,74.228,1.929
C02307=1010.964,284.977,-148.910,-12.991,74.170,1.542
C02308=1010.995,284.781,-148.836,-13.237,74.123,1.164
C02309=1011.027,284.584,-148.763,-13.486,74.067,0.788
C02310=1011.058,284.387,-148.690,-13.735,74.009,0.411
C02311=1011.089,284.190,-148.618,-13.972,73.960,0.045
C02312=1011.119,283.993,-148.546,-14.214,73.900,-0.323
///RCONF 0,0,0,0,1,0,0,0,0,0,0,0,0,0,0,0,0,0,0,0,0,0,0,0
C02313=1011.149,283.797,-148.474,-14.449,73.848,-0.686
C02314=1011.208,283.402,-148.334,-14.919,73.727,-1.405
C02315=1011.265,283.007,-148.194,-15.367,73.620,-2.105
C02316=1011.322,282.612,-148.056,-15.803,73.514,-2.791
C02317=1011.377,282.216,-147.919,-16.231,73.405,-3.467
C02318=1011.432,281.819,-147.784,-16.645,73.298,-4.127
C02319=1011.485,281.422,-147.652,-17.057,73.182,-4.782
C02320=1011.537,281.027,-147.520,-17.446,73.083,-5.416
C02321=1011.588,280.629,-147.391,-17.831,72.977,-6.042
C02322=1011.637,280.230,-147.262,-18.206,72.869,-6.656
C02323=1011.685,279.833,-147.136,-18.572,72.762,-7.259
C02324=1011.733,279.435,-147.011,-18.924,72.665,-7.849
C02325=1011.779,279.035,-146.888,-19.272,72.559,-8.431
C02326=1011.824,278.636,-146.765,-19.605,72.472,-9.001
C02327=1011.868,278.237,-146.645,-19.937,72.373,-9.566
C02328=1011.911,277.837,-146.527,-20.268,72.257,-10.128
C02329=1011.952,277.438,-146.409,-20.578,72.179,-10.673
C02330=1011.994,277.037,-146.294,-20.894,72.073,-11.219
C02331=1012.032,276.637,-146.180,-21.198,71.980,-11.755
C02332=1012.071,276.236,-146.067,-21.499,71.880,-12.286
C02333=1012.108,275.835,-145.957,-21.792,71.783,-12.807
C02334=1012.146,275.434,-145.847,-22.081,71.686,-13.326
C02335=1012.180,275.032,-145.739,-22.361,71.598,-13.834
C02336=1012.215,274.630,-145.633,-22.638,71.504,-14.338
C02337=1012.249,274.228,-145.528,-22.912,71.399,-14.837
C02338=1012.280,273.826,-145.425,-23.177,71.309,-15.328
C02339=1012.312,273.424,-145.322,-23.438,71.220,-15.814
C02340=1012.341,273.021,-145.222,-23.692,71.138,-16.294
C02341=1012.371,272.618,-145.124,-23.948,71.022,-16.770
C02342=1012.398,272.215,-145.026,-24.192,70.943,-17.238
C02343=1012.425,271.812,-144.930,-24.436,70.847,-17.702
C02344=1012.452,271.408,-144.836,-24.675,70.755,-18.163
C02345=1012.477,271.004,-144.742,-24.910,70.676,-18.621
C02346=1012.501,270.600,-144.652,-25.142,70.571,-19.073
C02347=1012.523,270.197,-144.561,-25.368,70.505,-19.521
C02348=1012.546,269.793,-144.472,-25.593,70.406,-19.965
C02349=1012.566,269.388,-144.385,-25.814,70.326,-20.408
C02350=1012.587,268.984,-144.300,-26.031,70.212,-20.843
C02351=1012.605,268.579,-144.215,-26.245,70.134,-21.276
C02352=1012.623,268.174,-144.132,-26.455,70.052,-21.706
C02353=1012.640,267.769,-144.051,-26.662,69.950,-22.130
C02354=1012.656,267.364,-143.970,-26.867,69.885,-22.554
C02355=1012.670,266.959,-143.892,-27.068,69.787,-22.973
C02356=1012.685,266.553,-143.815,-27.265,69.704,-23.388
C02357=1012.698,266.148,-143.740,-27.461,69.629,-23.802
C02358=1012.710,265.742,-143.665,-27.653,69.543,-24.210
C02359=1012.721,265.336,-143.592,-27.842,69.445,-24.615
C02360=1012.731,264.929,-143.522,-28.027,69.352,-25.016
C02361=1012.739,264.523,-143.450,-28.214,69.295,-25.420
C02362=1012.748,264.117,-143.382,-28.393,69.186,-25.814
C02363=1012.755,263.711,-143.315,-28.572,69.104,-26.208
C02364=1012.762,263.304,-143.249,-28.751,69.038,-26.603
C02365=1012.767,262.898,-143.185,-28.922,68.938,-26.989
C02366=1012.771,262.491,-143.122,-29.097,68.876,-27.379
C02367=1012.774,262.085,-143.060,-29.265,68.783,-27.762
C02368=1012.776,261.677,-143.000,-29.434,68.712,-28.144
C02369=1012.779,261.271,-142.942,-29.594,68.602,-28.519
C02370=1012.779,260.863,-142.885,-29.758,68.528,-28.896
C02371=1012.777,260.456,-142.828,-29.919,68.451,-29.272
C02372=1012.777,260.049,-142.775,-30.074,68.355,-29.640
C02373=1012.774,259.642,-142.721,-30.235,68.294,-30.012
C02374=1012.761,258.410,-142.568,-30.692,68.063,-31.105
C02375=1012.758,258.165,-142.539,-30.688,68.053,-31.100
C02376=1012.754,257.920,-142.510,-30.686,68.042,-31.098
C02377=1012.751,257.674,-142.481,-30.682,68.032,-31.094
C02378=1012.748,257.429,-142.452,-30.680,68.022,-31.092
C02379=1012.744,257.184,-142.423,-30.677,68.012,-31.089
C02380=1012.741,256.939,-142.394,-30.675,68.003,-31.086
C02381=1012.737,256.694,-142.365,-30.672,67.993,-31.083
C02382=1012.734,256.448,-142.337,-30.669,67.985,-31.081
C02383=1012.731,256.203,-142.308,-30.667,67.976,-31.079
C02384=1012.728,255.958,-142.278,-30.664,67.968,-31.075
C02385=1012.725,255.713,-142.250,-30.662,67.959,-31.073
C02386=1012.721,255.468,-142.221,-30.660,67.948,-31.071
C02387=1012.718,255.223,-142.192,-30.656,67.938,-31.066
C02388=1012.715,254.977,-142.164,-30.654,67.927,-31.064
C02389=1012.711,254.732,-142.135,-30.651,67.918,-31.061
C02390=1012.707,254.487,-142.106,-30.648,67.908,-31.058
C02391=1012.705,254.241,-142.076,-30.645,67.897,-31.056
C02392=1012.701,253.996,-142.047,-30.643,67.889,-31.052
C02393=1012.698,253.751,-142.019,-30.640,67.881,-31.050
C02394=1012.695,253.506,-141.990,-30.638,67.872,-31.048
C02395=1012.691,253.261,-141.961,-30.636,67.863,-31.046
C02396=1012.688,253.016,-141.932,-30.633,67.853,-31.042
C02397=1012.685,252.770,-141.904,-30.630,67.842,-31.039
C02398=1012.682,252.525,-141.875,-30.627,67.832,-31.036
C02399=1012.679,252.280,-141.847,-30.625,67.822,-31.034
C02400=1012.675,252.035,-141.818,-30.621,67.811,-31.030
C02401=1012.672,251.790,-141.789,-30.619,67.802,-31.028
C02402=1012.669,251.544,-141.761,-30.616,67.793,-31.024
C02403=1012.666,251.300,-141.732,-30.614,67.784,-31.022
C02404=1012.663,251.054,-141.704,-30.611,67.774,-31.019
C02405=1012.660,250.809,-141.674,-30.609,67.765,-31.017
C02406=1012.657,250.564,-141.646,-30.606,67.757,-31.013
C02407=1012.654,250.318,-141.617,-30.604,67.747,-31.011
C02408=1012.650,250.073,-141.588,-30.601,67.736,-31.008
C02409=1012.647,249.828,-141.560,-30.598,67.726,-31.005
C02410=1012.644,249.583,-141.531,-30.595,67.715,-31.002
C02411=1012.641,249.337,-141.503,-30.592,67.705,-30.999
C02412=1012.637,249.092,-141.474,-30.589,67.695,-30.995
C02413=1012.635,248.846,-141.446,-30.587,67.686,-30.995
C02414=1012.631,248.601,-141.417,-30.585,67.676,-30.992
C02415=1012.628,248.356,-141.389,-30.582,67.668,-30.988
C02416=1012.626,248.111,-141.361,-30.580,67.659,-30.986
C02417=1012.622,247.866,-141.332,-30.577,67.650,-30.984
C02418=1012.619,247.620,-141.304,-30.574,67.639,-30.981
C02419=1012.616,247.375,-141.275,-30.571,67.628,-30.976
C02420=1012.613,247.130,-141.247,-30.569,67.618,-30.975
C02421=1012.610,246.884,-141.218,-30.566,67.607,-30.973
C02422=1012.607,246.639,-141.189,-30.563,67.597,-30.969
C02423=1012.604,246.394,-141.161,-30.561,67.588,-30.967
C02424=1012.601,246.148,-141.133,-30.558,67.578,-30.963
C02425=1012.598,245.903,-141.104,-30.555,67.569,-30.960
C02426=1012.595,245.658,-141.076,-30.553,67.560,-30.958
C02427=1012.592,245.412,-141.048,-30.551,67.551,-30.956
C02428=1012.589,245.167,-141.020,-30.548,67.541,-30.953
C02429=1012.586,244.922,-140.991,-30.545,67.530,-30.950
C02430=1012.583,244.676,-140.962,-30.543,67.519,-30.948
C02431=1012.580,244.431,-140.934,-30.539,67.509,-30.944
C02432=1012.577,244.185,-140.906,-30.537,67.498,-30.942
C02433=1012.575,243.940,-140.878,-30.534,67.489,-30.939
C02434=1012.571,243.695,-140.849,-30.532,67.479,-30.936
C02435=1012.568,243.450,-140.821,-30.529,67.469,-30.933
C02436=1012.565,243.204,-140.793,-30.526,67.460,-30.929
C02437=1012.562,242.959,-140.765,-30.524,67.451,-30.927
C02438=1012.560,242.713,-140.736,-30.522,67.442,-30.925
C02439=1012.557,242.468,-140.708,-30.519,67.431,-30.924
C02440=1012.554,242.223,-140.679,-30.516,67.421,-30.919
C02441=1012.551,241.978,-140.652,-30.513,67.410,-30.917
C02442=1012.548,241.732,-140.623,-30.511,67.399,-30.915
C02443=1012.545,241.487,-140.595,-30.508,67.389,-30.911
C02444=1012.542,241.241,-140.567,-30.505,67.378,-30.909
C02445=1012.539,240.996,-140.539,-30.503,67.369,-30.906
C02446=1012.537,240.750,-140.511,-30.500,67.359,-30.903
C02447=1012.534,240.505,-140.482,-30.498,67.350,-30.901
C02448=1012.531,240.260,-140.455,-30.495,67.340,-30.898
C02449=1012.528,240.014,-140.426,-30.493,67.331,-30.896
C02450=1012.525,239.769,-140.398,-30.490,67.320,-30.893
C02451=1012.522,239.524,-140.370,-30.487,67.310,-30.888
C02452=1012.519,239.278,-140.342,-30.484,67.299,-30.887
C02453=1012.516,239.032,-140.314,-30.482,67.288,-30.884
C02454=1012.514,238.788,-140.286,-30.479,67.278,-30.881
C02455=1012.511,238.542,-140.258,-30.477,67.268,-30.879
C02456=1012.508,238.295,-140.230,-30.474,67.258,-30.876
C02457=1012.506,238.051,-140.202,-30.471,67.248,-30.873
C02458=1012.503,237.805,-140.174,-30.469,67.239,-30.870
C02459=1012.500,237.559,-140.146,-30.466,67.230,-30.868
C02460=1012.497,237.314,-140.118,-30.464,67.220,-30.865
C02461=1012.494,237.069,-140.090,-30.461,67.209,-30.862
C02462=1012.492,236.824,-140.062,-30.458,67.197,-30.860
C02463=1012.489,236.578,-140.035,-30.456,67.188,-30.856
C02464=1012.486,236.332,-140.006,-30.453,67.176,-30.854
C02465=1012.484,236.087,-139.978,-30.451,67.166,-30.852
C02466=1012.481,235.841,-139.950,-30.448,67.156,-30.849
C02467=1012.478,235.596,-139.922,-30.445,67.147,-30.846
C02468=1012.475,235.350,-139.895,-30.442,67.137,-30.843
C02469=1012.472,235.105,-139.867,-30.440,67.127,-30.840
C02470=1012.470,234.860,-139.839,-30.438,67.118,-30.838
C02471=1012.467,234.614,-139.811,-30.435,67.107,-30.835
C02472=1012.465,234.368,-139.783,-30.432,67.096,-30.833
C02473=1012.462,234.123,-139.755,-30.430,67.086,-30.830
C02474=1012.460,233.878,-139.727,-30.427,67.075,-30.827
C02475=1012.457,233.632,-139.699,-30.424,67.063,-30.824
C02476=1012.454,233.387,-139.672,-30.421,67.054,-30.821
C02477=1012.451,233.140,-139.644,-30.419,67.043,-30.820
C02478=1012.448,232.895,-139.616,-30.417,67.033,-30.817
C02479=1012.446,232.650,-139.588,-30.414,67.024,-30.814
C02480=1012.444,232.403,-139.560,-30.411,67.014,-30.811
C02481=1012.441,232.159,-139.532,-30.409,67.004,-30.808
C02482=1012.438,231.913,-139.504,-30.407,66.994,-30.806
C02483=1012.436,231.667,-139.477,-30.404,66.982,-30.803
C02484=1012.433,231.422,-139.449,-30.401,66.971,-30.801
C02485=1012.431,231.176,-139.422,-30.398,66.961,-30.797
C02486=1012.428,230.931,-139.394,-30.396,66.950,-30.795
C02487=1012.425,230.685,-139.367,-30.393,66.939,-30.793
C02488=1012.423,230.439,-139.338,-30.390,66.929,-30.790
C02489=1012.421,230.194,-139.311,-30.388,66.919,-30.787
C02490=1012.418,229.949,-139.283,-30.385,66.910,-30.784
C02491=1012.415,229.703,-139.256,-30.383,66.899,-30.782
C02492=1012.413,229.458,-139.228,-30.381,66.890,-30.780
C02493=1012.410,229.212,-139.200,-30.378,66.878,-30.777
C02494=1012.408,228.967,-139.172,-30.375,66.867,-30.774
C02495=1012.405,228.720,-139.145,-30.372,66.856,-30.770
C02496=1012.403,228.475,-139.117,-30.370,66.846,-30.768
C02497=1012.400,228.229,-139.089,-30.367,66.835,-30.766
C02498=1012.398,227.983,-139.062,-30.365,66.825,-30.763
C02499=1012.396,227.738,-139.035,-30.362,66.814,-30.760
C02500=1012.393,227.492,-139.007,-30.359,66.804,-30.757
C02501=1012.390,227.247,-138.980,-30.357,66.794,-30.754
C02502=1012.387,227.001,-138.952,-30.355,66.785,-30.753
C02503=1012.386,226.755,-138.924,-30.352,66.774,-30.750
C02504=1012.383,226.509,-138.896,-30.349,66.763,-30.747
C02505=1012.381,226.264,-138.869,-30.347,66.751,-30.745
C02506=1012.378,226.019,-138.842,-30.344,66.740,-30.742
C02507=1012.376,225.773,-138.814,-30.341,66.730,-30.739
C02508=1012.373,225.527,-138.787,-30.339,66.719,-30.737
C02509=1012.371,225.282,-138.759,-30.336,66.708,-30.734
C02510=1012.369,225.036,-138.731,-30.334,66.698,-30.732
C02511=1012.367,224.790,-138.704,-30.331,66.688,-30.729
C02512=1012.364,224.545,-138.677,-30.329,66.678,-30.727
C02513=1012.361,224.299,-138.649,-30.326,66.668,-30.724
C02514=1012.359,224.053,-138.622,-30.324,66.658,-30.721
C02515=1012.356,223.807,-138.594,-30.321,66.646,-30.718
C02516=1012.354,223.562,-138.567,-30.318,66.635,-30.715
C02517=1012.353,223.316,-138.539,-30.316,66.623,-30.713
C02518=1012.350,223.070,-138.512,-30.313,66.613,-30.711
C02519=1012.348,222.824,-138.485,-30.311,66.602,-30.709
C02520=1012.345,222.579,-138.457,-30.308,66.592,-30.706
C02521=1012.342,222.333,-138.430,-30.306,66.580,-30.704
C02522=1012.340,222.088,-138.403,-30.303,66.571,-30.701
C02523=1012.339,221.842,-138.375,-30.301,66.561,-30.698
C02524=1012.336,221.595,-138.347,-30.299,66.551,-30.696
C02525=1012.334,221.350,-138.320,-30.296,66.541,-30.694
C02526=1012.331,221.104,-138.293,-30.294,66.529,-30.691
C02527=1012.329,220.859,-138.266,-30.291,66.518,-30.689
C02528=1012.326,220.613,-138.239,-30.288,66.508,-30.686
C02529=1012.324,220.368,-138.211,-30.286,66.497,-30.683
C02530=1012.322,220.118,-138.183,-30.284,66.487,-30.682
C02531=1012.319,219.858,-138.155,-30.282,66.474,-30.681
C02532=1012.318,219.586,-138.124,-30.279,66.463,-30.679
C02533=1012.315,219.305,-138.093,-30.276,66.451,-30.675
C02534=1012.312,219.008,-138.061,-30.273,66.437,-30.672
C02535=1012.309,218.705,-138.026,-30.269,66.424,-30.667
C02536=1012.307,218.409,-137.994,-30.266,66.411,-30.663
C02537=1012.304,218.115,-137.961,-30.262,66.398,-30.658
C02538=1012.301,217.826,-137.930,-30.259,66.386,-30.655
C02539=1012.299,217.545,-137.899,-30.256,66.374,-30.651
C02540=1012.296,217.281,-137.869,-30.254,66.362,-30.650
C02541=1012.294,217.022,-137.840,-30.251,66.351,-30.648
C02542=1012.293,216.767,-137.812,-30.249,66.338,-30.647
C02543=1012.290,216.519,-137.785,-30.247,66.327,-30.645
C02544=1012.287,216.273,-137.757,-30.244,66.317,-30.641
C02545=1012.285,216.027,-137.730,-30.242,66.306,-30.639
C02546=1012.283,215.781,-137.703,-30.239,66.295,-30.637
C02547=1012.281,215.536,-137.676,-30.237,66.283,-30.635
C02548=1012.279,215.291,-137.649,-30.234,66.273,-30.631
C02549=1012.277,215.046,-137.622,-30.232,66.262,-30.630
C02550=1012.275,214.800,-137.595,-30.229,66.251,-30.627
C02551=1012.273,214.555,-137.568,-30.227,66.239,-30.625
C02552=1012.271,214.311,-137.541,-30.224,66.229,-30.621
C02553=1012.268,214.066,-137.515,-30.222,66.218,-30.620
C02554=1012.266,213.822,-137.487,-30.219,66.207,-30.617
C02555=1012.265,213.578,-137.461,-30.217,66.196,-30.615
C02556=1012.263,213.334,-137.434,-30.214,66.185,-30.611
C02557=1012.260,213.090,-137.407,-30.212,66.175,-30.610
C02558=1012.259,212.847,-137.380,-30.209,66.163,-30.608
C02559=1012.256,212.603,-137.353,-30.207,66.152,-30.605
C02560=1012.254,212.360,-137.327,-30.204,66.142,-30.603
C02561=1012.252,212.116,-137.300,-30.202,66.131,-30.600
C02562=1012.251,211.873,-137.273,-30.199,66.119,-30.598
C02563=1012.249,211.630,-137.247,-30.197,66.108,-30.596
C02564=1012.246,211.387,-137.219,-30.194,66.098,-30.593
C02565=1012.245,211.145,-137.193,-30.192,66.087,-30.591
C02566=1012.243,210.902,-137.167,-30.190,66.076,-30.588
C02567=1012.241,210.660,-137.140,-30.187,66.064,-30.586
C02568=1012.239,210.417,-137.114,-30.185,66.054,-30.585
C02569=1012.236,210.175,-137.087,-30.183,66.042,-30.583
C02570=1012.234,209.932,-137.061,-30.180,66.031,-30.580
C02571=1012.233,209.690,-137.034,-30.177,66.021,-30.576
C02572=1012.230,209.447,-137.008,-30.175,66.010,-30.575
C02573=1012.229,209.205,-136.981,-30.173,65.999,-30.573
C02574=1012.227,208.963,-136.955,-30.171,65.987,-30.571
C02575=1012.225,208.720,-136.928,-30.168,65.976,-30.569
C02576=1012.223,208.478,-136.901,-30.166,65.965,-30.567
C02577=1012.221,208.235,-136.875,-30.163,65.955,-30.564
C02578=1012.220,207.993,-136.848,-30.161,65.943,-30.561
C02579=1012.218,207.750,-136.822,-30.158,65.932,-30.559
C02580=1012.215,207.508,-136.796,-30.157,65.921,-30.558
C02581=1012.214,207.264,-136.769,-30.154,65.910,-30.556
C02582=1012.212,207.021,-136.743,-30.152,65.899,-30.553
C02583=1012.210,206.779,-136.716,-30.149,65.887,-30.551
C02584=1012.208,206.536,-136.689,-30.146,65.877,-30.547
C02585=1012.206,206.292,-136.663,-30.144,65.865,-30.545
C02586=1012.204,206.049,-136.637,-30.142,65.855,-30.544
C02587=1012.202,205.806,-136.611,-30.140,65.843,-30.542
C02588=1012.201,205.563,-136.583,-30.137,65.832,-30.540
C02589=1012.199,205.318,-136.557,-30.135,65.821,-30.538
C02590=1012.197,205.075,-136.530,-30.133,65.809,-30.535
C02591=1012.195,204.830,-136.504,-30.130,65.798,-30.533
C02592=1012.194,204.587,-136.477,-30.128,65.787,-30.531
C02593=1012.191,204.342,-136.451,-30.125,65.775,-30.529
C02594=1012.190,204.097,-136.424,-30.122,65.765,-30.525
C02595=1012.188,203.854,-136.398,-30.120,65.753,-30.523
C02596=1012.186,203.609,-136.372,-30.118,65.742,-30.521
C02597=1012.185,203.362,-136.344,-30.115,65.731,-30.518
C02598=1012.181,202.116,-136.207,-29.776,65.826,-29.650
C02599=1012.181,201.897,-136.184,-29.775,65.815,-29.649
C02600=1012.181,201.487,-136.140,-29.771,65.795,-29.646
C02601=1012.182,201.276,-136.117,-29.769,65.784,-29.645
C02602=1012.183,201.059,-136.094,-29.768,65.773,-29.644
C02603=1012.183,200.835,-136.069,-29.766,65.763,-29.643
C02604=1012.183,200.597,-136.043,-29.764,65.751,-29.641
C02605=1012.184,200.342,-136.016,-29.763,65.739,-29.641
C02606=1012.184,200.088,-135.988,-29.760,65.726,-29.639
C02607=1012.184,199.847,-135.962,-29.758,65.715,-29.637
C02608=1012.185,199.615,-135.938,-29.757,65.703,-29.638
C02609=1012.186,199.385,-135.913,-29.755,65.692,-29.636
C02610=1012.186,199.143,-135.887,-29.753,65.680,-29.634
C02611=1012.186,198.752,-135.844,-29.750,65.662,-29.633
C02612=1012.187,198.361,-135.803,-29.747,65.642,-29.631
C02613=1012.187,198.114,-135.776,-29.746,65.630,-29.631
C02614=1012.188,197.878,-135.751,-29.744,65.618,-29.629
C02615=1012.189,197.643,-135.725,-29.742,65.606,-29.628
C02616=1012.189,197.407,-135.700,-29.740,65.595,-29.626
C02617=1012.190,197.171,-135.674,-29.738,65.582,-29.626
C02618=1012.190,196.935,-135.649,-29.737,65.572,-29.625
C02619=1012.191,196.699,-135.624,-29.735,65.560,-29.623
C02620=1012.190,196.463,-135.599,-29.733,65.550,-29.623
C02621=1012.191,196.227,-135.573,-29.732,65.539,-29.622
C02622=1012.191,195.991,-135.548,-29.730,65.528,-29.620
C02623=1012.192,195.755,-135.523,-29.729,65.516,-29.621
C02624=1012.193,195.519,-135.498,-29.727,65.505,-29.619
C02625=1012.193,195.283,-135.472,-29.725,65.492,-29.618
C02626=1012.194,195.047,-135.447,-29.723,65.481,-29.617
C02627=1012.194,194.811,-135.421,-29.721,65.469,-29.616
C02628=1012.195,194.575,-135.396,-29.720,65.458,-29.615
C02629=1012.195,194.340,-135.371,-29.718,65.447,-29.614
C02630=1012.195,194.104,-135.346,-29.716,65.436,-29.613
C02631=1012.196,193.868,-135.320,-29.715,65.425,-29.612
C02632=1012.196,193.632,-135.295,-29.713,65.415,-29.611
C02633=1012.197,193.395,-135.270,-29.712,65.402,-29.611
C02634=1012.198,193.159,-135.245,-29.710,65.391,-29.609
C02635=1012.199,192.924,-135.220,-29.709,65.380,-29.610
C02636=1012.199,192.688,-135.194,-29.707,65.368,-29.608
C02637=1012.199,192.452,-135.169,-29.705,65.357,-29.606
C02638=1012.199,192.216,-135.144,-29.704,65.345,-29.607
C02639=1012.200,191.981,-135.118,-29.702,65.335,-29.606
C02640=1012.201,191.744,-135.094,-29.701,65.324,-29.605
C02641=1012.202,191.509,-135.069,-29.699,65.313,-29.605
C02642=1012.202,191.273,-135.043,-29.697,65.303,-29.604
C02643=1012.203,191.037,-135.018,-29.696,65.290,-29.604
C02644=1012.203,190.801,-134.992,-29.694,65.279,-29.602
C02645=1012.203,190.565,-134.967,-29.692,65.267,-29.601
C02646=1012.204,190.329,-134.943,-29.691,65.256,-29.601
C02647=1012.205,190.093,-134.917,-29.689,65.245,-29.599
C02648=1012.205,189.857,-134.892,-29.687,65.234,-29.598
C02649=1012.206,189.621,-134.867,-29.686,65.222,-29.599
C02650=1012.207,189.386,-134.841,-29.685,65.212,-29.598
C02651=1012.207,189.150,-134.817,-29.683,65.201,-29.598
C02652=1012.207,188.914,-134.792,-29.682,65.190,-29.597
C02653=1012.208,188.678,-134.766,-29.680,65.179,-29.595
C02654=1012.209,188.443,-134.741,-29.679,65.168,-29.596
C02655=1012.210,188.206,-134.717,-29.677,65.156,-29.594
C02656=1012.210,187.970,-134.691,-29.675,65.145,-29.593
C02657=1012.210,187.734,-134.666,-29.674,65.133,-29.593
C02658=1012.211,187.499,-134.641,-29.672,65.123,-29.592
C02659=1012.212,187.263,-134.616,-29.671,65.112,-29.592
C02660=1012.212,187.027,-134.591,-29.669,65.101,-29.591
C02661=1012.213,186.791,-134.566,-29.668,65.091,-29.590
C02662=1012.214,186.555,-134.540,-29.667,65.081,-29.591
C02663=1012.214,186.319,-134.516,-29.665,65.068,-29.590
C02664=1012.215,186.084,-134.491,-29.664,65.057,-29.589
C02665=1012.215,185.848,-134.466,-29.663,65.045,-29.589
C02666=1012.216,185.611,-134.441,-29.661,65.035,-29.589
C02667=1012.217,185.376,-134.416,-29.659,65.023,-29.587
C02668=1012.217,185.140,-134.391,-29.658,65.013,-29.586
C02669=1012.217,184.904,-134.366,-29.656,65.002,-29.586
C02670=1012.219,184.669,-134.341,-29.655,64.991,-29.585
C02671=1012.219,184.433,-134.316,-29.654,64.982,-29.585
C02672=1012.220,184.197,-134.290,-29.652,64.971,-29.585
C02673=1012.220,183.961,-134.266,-29.651,64.959,-29.584
C02674=1012.221,183.725,-134.241,-29.649,64.948,-29.584
C02675=1012.222,183.490,-134.216,-29.648,64.936,-29.585
C02676=1012.223,183.253,-134.191,-29.646,64.925,-29.583
C02677=1012.222,183.018,-134.166,-29.645,64.914,-29.582
C02678=1012.223,182.782,-134.141,-29.643,64.904,-29.581
C02679=1012.224,182.546,-134.117,-29.642,64.893,-29.581
C02680=1012.225,182.310,-134.091,-29.641,64.883,-29.581
C02681=1012.226,182.074,-134.066,-29.640,64.873,-29.581
C02682=1012.226,181.839,-134.042,-29.639,64.861,-29.581
C02683=1012.227,181.603,-134.017,-29.637,64.850,-29.581
C02684=1012.227,181.367,-133.991,-29.635,64.839,-29.579
C02685=1012.229,181.131,-133.967,-29.634,64.827,-29.580
C02686=1012.228,180.895,-133.942,-29.633,64.817,-29.579
C02687=1012.230,180.660,-133.917,-29.631,64.806,-29.579
C02688=1012.230,180.424,-133.892,-29.630,64.795,-29.578
C02689=1012.231,180.188,-133.867,-29.629,64.786,-29.578
C02690=1012.231,179.952,-133.843,-29.627,64.775,-29.578
C02691=1012.233,179.717,-133.818,-29.626,64.764,-29.577
C02692=1012.233,179.481,-133.792,-29.625,64.754,-29.576
C02693=1012.234,179.245,-133.768,-29.624,64.742,-29.577
C02694=1012.234,179.009,-133.743,-29.622,64.731,-29.577
C02695=1012.235,178.774,-133.718,-29.621,64.720,-29.578
C02696=1012.236,178.537,-133.693,-29.620,64.709,-29.577
C02697=1012.236,178.302,-133.669,-29.618,64.699,-29.576
C02698=1012.237,178.066,-133.644,-29.617,64.688,-29.576
C02699=1012.238,177.831,-133.619,-29.616,64.678,-29.576
C02700=1012.239,177.595,-133.594,-29.615,64.667,-29.576
C02701=1012.239,177.359,-133.570,-29.614,64.658,-29.576
C02702=1012.240,177.124,-133.545,-29.612,64.647,-29.575
C02703=1012.241,176.887,-133.520,-29.611,64.636,-29.575
C02704=1012.241,176.652,-133.495,-29.609,64.624,-29.575
C02705=1012.242,176.416,-133.471,-29.608,64.613,-29.574
C02706=1012.243,176.180,-133.446,-29.607,64.603,-29.574
C02707=1012.244,175.945,-133.422,-29.605,64.593,-29.574
C02708=1012.244,175.709,-133.396,-29.604,64.582,-29.573
C02709=1012.246,175.474,-133.371,-29.603,64.572,-29.574
C02710=1012.246,175.237,-133.347,-29.602,64.561,-29.573
C02711=1012.247,175.002,-133.322,-29.601,64.552,-29.574
C02712=1012.248,174.766,-133.298,-29.599,64.541,-29.573
C02713=1012.249,174.530,-133.272,-29.598,64.529,-29.574
C02714=1012.249,174.295,-133.248,-29.597,64.519,-29.573
C02715=1012.250,174.059,-133.223,-29.596,64.508,-29.573
C02716=1012.250,173.823,-133.199,-29.595,64.497,-29.574
C02717=1012.251,173.588,-133.174,-29.594,64.487,-29.574
C02718=1012.252,173.353,-133.149,-29.592,64.476,-29.573
C02719=1012.252,173.116,-133.125,-29.591,64.466,-29.574
C02720=1012.254,172.881,-133.100,-29.590,64.455,-29.573
C02721=1012.255,172.645,-133.075,-29.589,64.446,-29.572
C02722=1012.255,172.410,-133.051,-29.588,64.435,-29.573
C02723=1012.256,172.174,-133.026,-29.586,64.424,-29.573
C02724=1012.257,171.938,-133.001,-29.585,64.414,-29.572
C02725=1012.258,171.703,-132.977,-29.584,64.404,-29.573
C02726=1012.258,171.467,-132.952,-29.583,64.392,-29.574
C02727=1012.259,171.231,-132.928,-29.582,64.382,-29.573
C02728=1012.260,170.996,-132.903,-29.581,64.372,-29.573
C02729=1012.261,170.760,-132.878,-29.580,64.362,-29.574
C02730=1012.261,170.525,-132.854,-29.578,64.352,-29.572
C02731=1012.262,170.289,-132.829,-29.577,64.342,-29.572
C02732=1012.264,170.053,-132.804,-29.576,64.331,-29.573
C02733=1012.264,169.817,-132.780,-29.575,64.321,-29.574
C02734=1012.265,169.582,-132.755,-29.574,64.310,-29.573
C02735=1012.265,169.346,-132.731,-29.572,64.299,-29.573
C02736=1012.266,169.111,-132.706,-29.571,64.289,-29.573
C02737=1012.267,168.875,-132.682,-29.570,64.279,-29.573
C02738=1012.267,168.640,-132.657,-29.569,64.269,-29.573
C02739=1012.269,168.404,-132.633,-29.568,64.259,-29.574
C02740=1012.269,168.169,-132.608,-29.567,64.249,-29.574
C02741=1012.271,167.933,-132.584,-29.566,64.238,-29.574
C02742=1012.271,167.698,-132.559,-29.565,64.229,-29.574
C02743=1012.272,167.462,-132.535,-29.564,64.217,-29.575
C02744=1012.272,167.226,-132.511,-29.563,64.206,-29.575
C02745=1012.273,166.990,-132.486,-29.562,64.196,-29.575
C02746=1012.275,166.755,-132.461,-29.560,64.186,-29.574
C02747=1012.275,166.520,-132.437,-29.559,64.176,-29.575
C02748=1012.277,166.284,-132.412,-29.559,64.166,-29.575
C02749=1012.277,166.049,-132.388,-29.558,64.156,-29.576
C02750=1012.278,165.813,-132.363,-29.556,64.147,-29.575
C02751=1012.278,165.577,-132.339,-29.555,64.136,-29.574
C02752=1012.279,165.341,-132.314,-29.554,64.127,-29.575
C02753=1012.280,165.106,-132.290,-29.553,64.116,-29.577
C02754=1012.281,164.804,-132.259,-29.552,64.103,-29.576
C02755=1012.282,164.485,-132.226,-29.550,64.090,-29.576
C02756=1012.284,164.097,-132.185,-29.549,64.073,-29.578
C02757=1012.285,163.877,-132.162,-29.548,64.063,-29.578
C02758=1012.285,163.656,-132.139,-29.547,64.054,-29.577
C02759=1012.287,163.419,-132.115,-29.546,64.044,-29.578
C02760=1012.288,163.156,-132.088,-29.545,64.033,-29.579
C02761=1012.288,162.862,-132.057,-29.544,64.020,-29.579
C02762=1012.289,162.554,-132.026,-29.542,64.006,-29.579
C02763=1012.290,162.262,-131.995,-29.541,63.994,-29.579
C02764=1012.291,161.956,-131.964,-29.539,63.982,-29.579
C02765=1012.292,161.653,-131.932,-29.539,63.968,-29.581
C02766=1012.294,161.360,-131.902,-29.537,63.956,-29.581
C02767=1012.294,161.082,-131.874,-29.536,63.944,-29.581
C02768=1012.296,160.820,-131.846,-29.535,63.931,-29.581
C02769=1012.296,160.570,-131.820,-29.534,63.922,-29.581
C02770=1012.297,160.330,-131.796,-29.532,63.911,-29.581
C02771=1012.298,160.096,-131.772,-29.531,63.901,-29.581
C02772=1012.300,159.864,-131.749,-29.526,63.844,-29.583
C02773=1012.303,159.631,-131.729,-29.514,63.733,-29.583
C02774=1012.306,159.397,-131.710,-29.501,63.621,-29.583
C02775=1012.308,159.161,-131.690,-29.489,63.509,-29.583
C02776=1012.311,158.924,-131.669,-29.477,63.396,-29.585
C02777=1012.313,158.689,-131.649,-29.465,63.284,-29.586
C02778=1012.318,158.275,-131.615,-29.444,63.088,-29.587
C02779=1012.322,157.982,-131.590,-29.430,62.948,-29.591
C02780=1012.325,157.745,-131.569,-29.418,62.835,-29.591
C02781=1012.327,157.507,-131.550,-29.407,62.722,-29.594
C02782=1012.330,157.268,-131.529,-29.396,62.609,-29.598
C02783=1012.333,157.030,-131.509,-29.385,62.496,-29.600
C02784=1012.336,156.789,-131.489,-29.373,62.383,-29.602
C02785=1012.338,156.551,-131.468,-29.362,62.269,-29.605
C02786=1012.341,156.311,-131.448,-29.351,62.156,-29.609
C02787=1012.344,156.072,-131.427,-29.340,62.042,-29.613
C02788=1012.347,155.832,-131.407,-29.330,61.929,-29.617
C02789=1012.350,155.593,-131.388,-29.319,61.816,-29.622
C02790=1012.353,155.354,-131.367,-29.308,61.703,-29.624
C02791=1012.355,155.114,-131.347,-29.298,61.590,-29.629
C02792=1012.359,154.874,-131.327,-29.287,61.476,-29.634
C02793=1012.361,154.634,-131.306,-29.277,61.363,-29.640
C02794=1012.365,154.393,-131.285,-29.267,61.249,-29.644
C02795=1012.367,154.152,-131.265,-29.256,61.136,-29.649
C02796=1012.370,153.910,-131.244,-29.246,61.023,-29.654
C02797=1012.373,153.669,-131.224,-29.236,60.910,-29.661
C02798=1012.376,153.428,-131.203,-29.226,60.796,-29.667
C02799=1012.379,153.187,-131.183,-29.216,60.683,-29.673
C02800=1012.382,152.945,-131.162,-29.206,60.570,-29.678
C02801=1012.385,152.703,-131.142,-29.196,60.457,-29.685
C02802=1012.387,152.461,-131.122,-29.187,60.343,-29.692
C02803=1012.391,152.218,-131.101,-29.177,60.230,-29.699
C02804=1012.394,151.969,-131.080,-29.167,60.114,-29.706
C02805=1012.397,151.715,-131.058,-29.157,59.994,-29.715
C02806=1012.400,151.451,-131.035,-29.147,59.872,-29.723
C02807=1012.404,151.180,-131.012,-29.136,59.746,-29.732
C02808=1012.407,150.902,-130.989,-29.126,59.617,-29.742
C02809=1012.411,150.615,-130.964,-29.115,59.484,-29.751
C02810=1012.415,150.322,-130.939,-29.104,59.348,-29.761
C02811=1012.418,150.026,-130.915,-29.093,59.211,-29.771
C02812=1012.422,149.727,-130.888,-29.081,59.072,-29.781
C02813=1012.426,149.426,-130.863,-29.070,58.934,-29.792
C02814=1012.430,149.126,-130.838,-29.059,58.795,-29.803
C02815=1012.433,148.830,-130.813,-29.048,58.659,-29.815
C02816=1012.438,148.539,-130.788,-29.038,58.524,-29.826
C02817=1012.441,148.253,-130.764,-29.028,58.393,-29.839
C02818=1012.445,147.976,-130.740,-29.018,58.265,-29.850
C02819=1012.448,147.706,-130.717,-29.008,58.141,-29.861
C02820=1012.451,147.444,-130.695,-28.999,58.020,-29.872
C02821=1012.455,147.190,-130.673,-28.990,57.904,-29.884
C02822=1012.457,146.942,-130.652,-28.981,57.790,-29.895
C02823=1012.461,146.698,-130.631,-28.973,57.679,-29.906
C02824=1012.464,146.456,-130.610,-28.964,57.567,-29.917
C02825=1012.467,146.213,-130.590,-28.956,57.458,-29.928
C02826=1012.470,145.971,-130.569,-28.948,57.347,-29.940
C02827=1012.475,145.617,-130.539,-28.936,57.185,-29.956
C02828=1012.480,145.245,-130.507,-28.923,57.016,-29.974
C02829=1012.483,145.003,-130.487,-28.915,56.907,-29.986
C02830=1012.486,144.762,-130.466,-28.907,56.796,-29.999
C02831=1012.489,144.521,-130.445,-28.899,56.687,-30.011
C02832=1012.493,144.279,-130.425,-28.891,56.578,-30.024
C02833=1012.495,144.039,-130.404,-28.883,56.469,-30.036
C02834=1012.499,143.798,-130.384,-28.875,56.360,-30.050
C02835=1012.502,143.557,-130.363,-28.867,56.252,-30.061
C02836=1012.505,143.317,-130.342,-28.859,56.143,-30.075
C02837=1012.508,143.076,-130.322,-28.852,56.035,-30.089
C02838=1012.512,142.836,-130.301,-28.844,55.927,-30.101
C02839=1012.515,142.597,-130.281,-28.836,55.819,-30.115
C02840=1012.518,142.357,-130.261,-28.828,55.711,-30.128
C02841=1012.521,142.118,-130.240,-28.820,55.604,-30.142
C02842=1012.524,141.878,-130.220,-28.812,55.496,-30.154
C02843=1012.528,141.640,-130.200,-28.805,55.390,-30.168
C02844=1012.531,141.394,-130.179,-28.797,55.279,-30.184
C02845=1012.534,141.183,-130.160,-28.790,55.185,-30.196
C02846=1012.538,140.928,-130.139,-28.782,55.071,-30.211
C02847=1012.541,140.635,-130.114,-28.773,54.941,-30.227
C02848=1012.545,140.383,-130.092,-28.765,54.829,-30.244
C02849=1012.548,140.109,-130.068,-28.756,54.706,-30.261
C02850=1012.552,139.813,-130.043,-28.747,54.575,-30.279
C02851=1012.556,139.504,-130.017,-28.737,54.439,-30.298
C02852=1012.560,139.192,-129.990,-28.728,54.300,-30.318
C02853=1012.565,138.884,-129.964,-28.718,54.164,-30.337
C02854=1012.569,138.590,-129.938,-28.709,54.033,-30.357
C02855=1012.573,138.316,-129.915,-28.700,53.912,-30.375
C02856=1012.576,138.064,-129.893,-28.692,53.801,-30.391
C02857=1012.581,137.644,-129.857,-28.679,53.616,-30.419
C02858=1012.587,137.260,-129.824,-28.668,53.447,-30.446
C02859=1012.593,136.843,-129.789,-28.655,53.265,-30.474
C02860=1012.597,136.460,-129.756,-28.643,53.097,-30.500
C02861=1012.603,136.074,-129.722,-28.631,52.928,-30.526
C02862=1012.610,135.655,-129.687,-28.618,52.746,-30.557
C02863=1012.612,135.430,-129.668,-28.611,52.648,-30.573
C02864=1012.615,135.197,-129.648,-28.604,52.546,-30.589
C02865=1012.619,134.912,-129.623,-28.595,52.422,-30.610
C02866=1012.623,134.616,-129.598,-28.586,52.294,-30.632
C02867=1012.626,134.377,-129.577,-28.579,52.190,-30.650
C02868=1012.629,134.142,-129.556,-28.572,52.089,-30.665
C02869=1012.633,133.907,-129.537,-28.564,51.987,-30.683
C02870=1012.637,133.671,-129.517,-28.557,51.886,-30.701
C02871=1012.639,133.436,-129.497,-28.550,51.784,-30.719
C02872=1012.643,133.201,-129.476,-28.543,51.682,-30.737
C02873=1012.646,132.966,-129.455,-28.536,51.581,-30.754
C02874=1012.649,132.731,-129.436,-28.528,51.480,-30.772
C02875=1012.653,132.496,-129.415,-28.521,51.379,-30.791
C02876=1012.656,132.261,-129.395,-28.514,51.279,-30.809
C02877=1012.659,132.017,-129.375,-28.507,51.175,-30.827
C02878=1012.663,131.786,-129.354,-28.500,51.076,-30.846
C02879=1012.666,131.554,-129.335,-28.492,50.977,-30.863
C02880=1012.669,131.319,-129.314,-28.485,50.876,-30.883
C02881=1012.672,131.085,-129.294,-28.478,50.776,-30.901
C02882=1012.676,130.849,-129.274,-28.471,50.676,-30.919
C02883=1012.679,130.614,-129.253,-28.464,50.576,-30.939
C02884=1012.682,130.379,-129.233,-28.456,50.476,-30.958
C02885=1012.685,130.144,-129.213,-28.449,50.377,-30.977
C02886=1012.689,129.909,-129.193,-28.442,50.277,-30.996
C02887=1012.692,129.674,-129.172,-28.435,50.178,-31.015
C02888=1012.695,129.439,-129.152,-28.427,50.078,-31.034
C02889=1012.698,129.204,-129.132,-28.420,49.979,-31.054
C02890=1012.702,128.968,-129.111,-28.413,49.880,-31.073
C02891=1012.706,128.734,-129.091,-28.406,49.781,-31.093
C02892=1012.708,128.499,-129.071,-28.398,49.682,-31.113
C02893=1012.712,128.263,-129.051,-28.391,49.582,-31.133
C02894=1012.715,128.028,-129.030,-28.384,49.484,-31.154
C02895=1012.718,127.793,-129.010,-28.377,49.385,-31.174
C02896=1012.722,127.558,-128.991,-28.369,49.287,-31.193
C02897=1012.725,127.323,-128.970,-28.362,49.188,-31.213
C02898=1012.729,127.087,-128.950,-28.355,49.091,-31.233
C02899=1012.731,126.852,-128.930,-28.347,48.993,-31.254
C02900=1012.735,126.617,-128.909,-28.340,48.894,-31.275
C02901=1012.739,126.382,-128.889,-28.333,48.797,-31.295
C02902=1012.742,126.147,-128.868,-28.325,48.700,-31.315
C02903=1012.745,125.912,-128.848,-28.318,48.601,-31.336
C02904=1012.748,125.677,-128.828,-28.311,48.505,-31.357
C02905=1012.752,125.442,-128.808,-28.303,48.408,-31.378
C02906=1012.755,125.207,-128.787,-28.296,48.310,-31.399
C02907=1012.758,124.972,-128.767,-28.288,48.213,-31.420
C02908=1012.761,124.737,-128.746,-28.281,48.116,-31.441
C02909=1012.764,124.502,-128.725,-28.274,48.020,-31.462
C02910=1012.768,124.267,-128.705,-28.266,47.923,-31.483
C02911=1012.772,124.032,-128.685,-28.259,47.826,-31.505
C02912=1012.774,123.797,-128.665,-28.251,47.731,-31.526
C02913=1012.778,123.562,-128.644,-28.244,47.634,-31.548
C02914=1012.782,123.327,-128.624,-28.236,47.538,-31.570
C02915=1012.785,123.092,-128.604,-28.229,47.442,-31.592
C02916=1012.788,122.857,-128.584,-28.221,47.347,-31.613
C02917=1012.791,122.621,-128.563,-28.214,47.251,-31.635
C02918=1012.795,122.387,-128.543,-28.206,47.155,-31.657
C02919=1012.798,122.151,-128.522,-28.199,47.061,-31.679
C02920=1012.802,121.916,-128.502,-28.191,46.965,-31.701
C02921=1012.804,121.681,-128.482,-28.184,46.871,-31.723
C02922=1012.808,121.446,-128.462,-28.176,46.776,-31.746
C02923=1012.812,121.211,-128.441,-28.169,46.682,-31.768
C02924=1012.815,120.976,-128.421,-28.161,46.588,-31.790
C02925=1012.817,120.741,-128.400,-28.153,46.494,-31.812
C02926=1012.822,120.506,-128.381,-28.145,46.394,-31.836
C02927=1012.825,120.271,-128.360,-28.137,46.291,-31.862
C02928=1012.829,120.036,-128.340,-28.128,46.188,-31.886
C02929=1012.832,119.801,-128.319,-28.120,46.085,-31.911
C02930=1012.836,119.567,-128.300,-28.112,45.983,-31.936
C02931=1012.839,119.331,-128.280,-28.103,45.882,-31.960
C02932=1012.843,119.095,-128.259,-28.095,45.780,-31.985
C02933=1012.847,118.861,-128.239,-28.086,45.677,-32.011
C02934=1012.850,118.626,-128.219,-28.078,45.575,-32.036
C02935=1012.853,118.391,-128.199,-28.069,45.474,-32.061
C02936=1012.857,118.155,-128.179,-28.061,45.373,-32.087
C02937=1012.862,117.820,-128.150,-28.048,45.229,-32.122
C02938=1012.868,117.451,-128.118,-28.035,45.069,-32.164
C02939=1012.871,117.215,-128.098,-28.026,44.969,-32.188
C02940=1012.875,116.981,-128.079,-28.017,44.868,-32.214
C02941=1012.878,116.745,-128.059,-28.009,44.768,-32.241
C02942=1012.882,116.511,-128.038,-28.000,44.668,-32.266
C02943=1012.886,116.275,-128.018,-27.991,44.568,-32.293
C02944=1012.890,116.041,-127.998,-27.983,44.467,-32.319
C02945=1012.893,115.805,-127.977,-27.974,44.368,-32.345
C02946=1012.896,115.571,-127.958,-27.965,44.268,-32.370
C02947=1012.900,115.335,-127.938,-27.956,44.168,-32.398
C02948=1012.903,115.100,-127.917,-27.948,44.070,-32.424
C02949=1012.907,114.865,-127.897,-27.939,43.971,-32.450
C02950=1012.911,114.630,-127.877,-27.930,43.871,-32.478
C02951=1012.915,114.395,-127.856,-27.921,43.772,-32.504
C02952=1012.917,114.160,-127.836,-27.912,43.674,-32.531
C02953=1012.921,113.926,-127.816,-27.903,43.575,-32.557
C02954=1012.925,113.690,-127.796,-27.894,43.477,-32.584
C02955=1012.929,113.455,-127.776,-27.885,43.379,-32.611
C02956=1012.932,113.220,-127.756,-27.876,43.281,-32.639
C02957=1012.936,112.985,-127.736,-27.867,43.183,-32.666
C02958=1012.939,112.750,-127.715,-27.858,43.086,-32.692
C02959=1012.943,112.516,-127.695,-27.849,42.989,-32.720
C02960=1012.946,112.280,-127.675,-27.840,42.891,-32.748
C02961=1012.949,112.045,-127.654,-27.831,42.794,-32.774
C02962=1012.953,111.810,-127.634,-27.822,42.697,-32.802
C02963=1012.957,111.574,-127.614,-27.812,42.599,-32.830
C02964=1012.961,111.340,-127.594,-27.803,42.503,-32.858
C02965=1012.964,111.105,-127.574,-27.794,42.407,-32.885
C02966=1012.968,110.870,-127.554,-27.785,42.310,-32.913
C02967=1012.971,110.635,-127.534,-27.776,42.214,-32.941
C02968=1012.974,110.400,-127.513,-27.766,42.118,-32.968
C02969=1012.978,110.165,-127.493,-27.757,42.023,-32.996
C02970=1012.982,109.930,-127.472,-27.748,41.926,-33.025
C02971=1012.986,109.695,-127.452,-27.738,41.831,-33.054
C02972=1012.989,109.460,-127.432,-27.729,41.735,-33.081
C02973=1012.993,109.225,-127.411,-27.719,41.640,-33.110
C02974=1012.996,108.990,-127.391,-27.710,41.545,-33.138
C02975=1012.999,108.755,-127.371,-27.701,41.451,-33.166
C02976=1013.003,108.520,-127.351,-27.691,41.356,-33.194
C02977=1013.006,108.285,-127.330,-27.681,41.261,-33.223
C02978=1013.011,108.050,-127.311,-27.672,41.167,-33.252
C02979=1013.014,107.814,-127.290,-27.662,41.073,-33.280
C02980=1013.017,107.579,-127.270,-27.653,40.979,-33.309
C02981=1013.021,107.345,-127.250,-27.643,40.886,-33.338
C02982=1013.025,107.109,-127.229,-27.633,40.791,-33.367
C02983=1013.029,106.875,-127.209,-27.624,40.699,-33.395
C02984=1013.031,106.640,-127.189,-27.614,40.605,-33.425
C02985=1013.035,106.404,-127.168,-27.604,40.511,-33.454
C02986=1013.038,106.170,-127.148,-27.595,40.419,-33.483
C02987=1013.042,105.934,-127.128,-27.585,40.326,-33.511
C02988=1013.046,105.700,-127.108,-27.575,40.233,-33.540
C02989=1013.049,105.464,-127.087,-27.565,40.141,-33.570
C02990=1013.053,105.229,-127.066,-27.555,40.048,-33.600
C02991=1013.057,104.995,-127.046,-27.546,39.956,-33.628
C02992=1013.060,104.759,-127.026,-27.536,39.865,-33.658
C02993=1013.063,104.524,-127.005,-27.526,39.773,-33.688
C02994=1013.066,104.290,-126.986,-27.516,39.681,-33.718
C02995=1013.070,104.054,-126.965,-27.506,39.590,-33.748
C02996=1013.073,103.819,-126.945,-27.496,39.498,-33.776
C02997=1013.077,103.584,-126.924,-27.486,39.407,-33.806
C02998=1013.083,103.213,-126.892,-27.470,39.263,-33.853
C02999=1013.088,102.879,-126.863,-27.456,39.135,-33.895
C03000=1013.091,102.644,-126.843,-27.446,39.044,-33.926
C03001=1013.095,102.409,-126.822,-27.436,38.955,-33.956
C03002=1013.099,102.174,-126.802,-27.425,38.865,-33.986
C03003=1013.102,101.939,-126.781,-27.415,38.775,-34.017
C03004=1013.105,101.704,-126.761,-27.405,38.685,-34.047
C03005=1013.108,101.469,-126.741,-27.395,38.595,-34.077
C03006=1013.112,101.234,-126.721,-27.384,38.505,-34.107
C03007=1013.115,100.998,-126.700,-27.374,38.417,-34.137
C03008=1013.119,100.763,-126.680,-27.364,38.328,-34.168
C03009=1013.123,100.528,-126.660,-27.353,38.240,-34.197
C03010=1013.126,100.293,-126.639,-27.343,38.151,-34.228
C03011=1013.129,100.058,-126.618,-27.333,38.062,-34.259
C03012=1013.133,99.823,-126.598,-27.322,37.973,-34.290
C03013=1013.137,99.588,-126.578,-27.312,37.885,-34.319
C03014=1013.140,99.353,-126.557,-27.301,37.798,-34.351
C03015=1013.143,99.118,-126.536,-27.291,37.710,-34.381
C03016=1013.146,98.884,-126.516,-27.280,37.622,-34.412
C03017=1013.150,98.648,-126.496,-27.270,37.535,-34.442
C03018=1013.153,98.413,-126.475,-27.259,37.448,-34.473
C03019=1013.156,98.178,-126.455,-27.249,37.361,-34.505
C03020=1013.160,97.942,-126.434,-27.238,37.274,-34.535
C03021=1013.164,97.708,-126.414,-27.227,37.187,-34.567
C03022=1013.167,97.472,-126.394,-27.217,37.100,-34.597
C03023=1013.170,97.237,-126.373,-27.206,37.014,-34.628
C03024=1013.174,97.002,-126.352,-27.195,36.928,-34.659
C03025=1013.178,96.767,-126.332,-27.185,36.842,-34.691
C03026=1013.181,96.532,-126.312,-27.174,36.756,-34.722
C03027=1013.184,96.297,-126.291,-27.163,36.671,-34.753
C03028=1013.188,96.061,-126.271,-27.152,36.585,-34.784
C03029=1013.190,95.826,-126.251,-27.141,36.500,-34.816
C03030=1013.194,95.591,-126.230,-27.131,36.416,-34.847
C03031=1013.197,95.357,-126.209,-27.120,36.329,-34.878
C03032=1013.201,95.122,-126.189,-27.109,36.245,-34.909
C03033=1013.204,94.886,-126.168,-27.098,36.161,-34.942
C03034=1013.208,94.651,-126.148,-27.087,36.076,-34.973
C03035=1013.211,94.416,-126.127,-27.076,35.992,-35.003
C03036=1013.214,94.180,-126.107,-27.065,35.908,-35.035
C03037=1013.218,93.945,-126.086,-27.054,35.825,-35.067
C03038=1013.222,93.711,-126.066,-27.043,35.741,-35.100
C03039=1013.225,93.475,-126.045,-27.032,35.657,-35.131
C03040=1013.228,93.240,-126.025,-27.021,35.575,-35.161
C03041=1013.232,93.005,-126.004,-27.010,35.491,-35.193
C03042=1013.235,92.769,-125.984,-26.998,35.409,-35.226
C03043=1013.238,92.534,-125.964,-26.987,35.325,-35.257
C03044=1013.241,92.300,-125.943,-26.976,35.243,-35.290
C03045=1013.244,92.064,-125.922,-26.965,35.161,-35.321
C03046=1013.247,91.829,-125.902,-26.954,35.078,-35.353
C03047=1013.251,91.594,-125.881,-26.942,34.997,-35.385
C03048=1013.255,91.359,-125.861,-26.931,34.914,-35.417
C03049=1013.258,91.124,-125.840,-26.920,34.833,-35.449
C03050=1013.262,90.888,-125.820,-26.909,34.751,-35.480
C03051=1013.265,90.629,-125.797,-26.896,34.662,-35.518
C03052=1013.269,90.310,-125.769,-26.881,34.552,-35.560
C03053=1013.274,89.976,-125.740,-26.865,34.437,-35.604
C03054=1013.278,89.693,-125.715,-26.851,34.341,-35.644
C03055=1013.281,89.456,-125.694,-26.839,34.259,-35.677
C03056=1013.285,89.224,-125.675,-26.828,34.180,-35.708
C03057=1013.288,88.994,-125.654,-26.817,34.103,-35.739
C03058=1013.291,88.767,-125.634,-26.806,34.026,-35.770
C03059=1013.294,88.543,-125.615,-26.795,33.950,-35.801
C03060=1013.297,88.319,-125.595,-26.784,33.875,-35.831
C03061=1013.301,88.095,-125.576,-26.773,33.799,-35.863
C03062=1013.304,87.871,-125.555,-26.762,33.724,-35.894
C03063=1013.306,87.644,-125.537,-26.751,33.648,-35.925
C03064=1013.309,87.413,-125.516,-26.739,33.572,-35.956
C03065=1013.313,87.179,-125.495,-26.728,33.493,-35.988
C03066=1013.316,86.944,-125.475,-26.716,33.415,-36.021
C03067=1013.321,86.546,-125.440,-26.696,33.284,-36.076
C03068=1013.325,86.228,-125.412,-26.681,33.179,-36.120
C03069=1013.329,85.989,-125.391,-26.669,33.101,-36.152
C03070=1013.332,85.749,-125.371,-26.657,33.022,-36.186
C03071=1013.335,85.509,-125.349,-26.645,32.944,-36.219
C03072=1013.339,85.269,-125.328,-26.633,32.866,-36.251
C03073=1013.342,85.028,-125.307,-26.621,32.787,-36.285
C03074=1013.345,84.786,-125.286,-26.609,32.709,-36.318
C03075=1013.349,84.544,-125.264,-26.597,32.630,-36.352
C03076=1013.352,84.302,-125.243,-26.585,32.553,-36.385
C03077=1013.355,84.059,-125.222,-26.572,32.474,-36.419
C03078=1013.358,83.816,-125.201,-26.560,32.396,-36.452
C03079=1013.362,83.572,-125.180,-26.548,32.319,-36.487
C03080=1013.365,83.328,-125.159,-26.536,32.241,-36.520
C03081=1013.369,83.083,-125.137,-26.523,32.163,-36.555
C03082=1013.371,82.837,-125.116,-26.511,32.086,-36.588
C03083=1013.375,82.592,-125.094,-26.499,32.008,-36.621
C03084=1013.378,82.346,-125.072,-26.486,31.930,-36.656
C03085=1013.381,82.100,-125.050,-26.474,31.853,-36.690
C03086=1013.384,81.854,-125.029,-26.461,31.776,-36.723
C03087=1013.387,81.606,-125.008,-26.449,31.699,-36.758
C03088=1013.392,81.360,-124.985,-26.436,31.622,-36.792
C03089=1013.394,81.117,-124.964,-26.424,31.547,-36.826
C03090=1013.398,80.889,-124.944,-26.412,31.476,-36.857
C03091=1013.400,80.671,-124.926,-26.401,31.409,-36.888
C03092=1013.402,80.454,-124.906,-26.390,31.342,-36.918
C03093=1013.406,80.226,-124.886,-26.378,31.272,-36.949
C03094=1013.409,79.983,-124.864,-26.366,31.198,-36.982
C03095=1013.413,79.737,-124.843,-26.353,31.123,-37.017
C03096=1013.416,79.492,-124.821,-26.341,31.048,-37.051
C03097=1013.419,79.250,-124.801,-26.328,30.974,-37.085
C03098=1013.422,79.011,-124.779,-26.316,30.902,-37.118
C03099=1013.425,78.774,-124.759,-26.304,30.831,-37.150
C03100=1013.428,78.539,-124.738,-26.292,30.760,-37.182
C03101=1013.430,78.307,-124.717,-26.280,30.690,-37.215
C03102=1013.434,78.077,-124.697,-26.268,30.622,-37.247
C03103=1013.437,77.849,-124.678,-26.256,30.554,-37.279
C03104=1013.439,77.620,-124.658,-26.245,30.486,-37.309
C03105=1013.443,77.393,-124.638,-26.233,30.418,-37.341
C03106=1013.446,77.166,-124.618,-26.221,30.352,-37.372
C03107=1013.448,76.937,-124.597,-26.209,30.283,-37.404
C03108=1013.452,76.707,-124.577,-26.197,30.216,-37.437
C03109=1013.454,76.474,-124.556,-26.185,30.148,-37.469
C03110=1013.457,76.239,-124.537,-26.173,30.079,-37.501
C03111=1013.460,76.002,-124.515,-26.161,30.009,-37.534
C03112=1013.463,75.760,-124.494,-26.148,29.939,-37.567
C03113=1013.466,75.517,-124.473,-26.136,29.869,-37.601
C03114=1013.469,75.271,-124.451,-26.123,29.798,-37.634
C03115=1013.472,75.024,-124.430,-26.110,29.727,-37.668
C03116=1013.476,74.775,-124.407,-26.097,29.656,-37.702
C03117=1013.479,74.516,-124.385,-26.084,29.582,-37.739
C03118=1013.482,74.245,-124.361,-26.070,29.504,-37.776
C03119=1013.486,73.977,-124.337,-26.056,29.428,-37.813
C03120=1013.488,73.726,-124.316,-26.043,29.357,-37.848
C03121=1013.491,73.481,-124.294,-26.030,29.287,-37.881
C03122=1013.495,73.235,-124.272,-26.017,29.218,-37.915
C03123=1013.498,72.990,-124.251,-26.004,29.150,-37.949
C03124=1013.500,72.746,-124.230,-25.992,29.082,-37.982
C03125=1013.504,72.503,-124.208,-25.979,29.013,-38.016
C03126=1013.506,72.260,-124.187,-25.966,28.946,-38.049
C03127=1013.510,72.018,-124.166,-25.954,28.880,-38.083
C03128=1013.512,71.776,-124.144,-25.941,28.813,-38.116
C03129=1013.516,71.535,-124.123,-25.929,28.747,-38.148
C03130=1013.518,71.293,-124.101,-25.916,28.680,-38.181
C03131=1013.521,71.052,-124.080,-25.904,28.615,-38.214
C03132=1013.524,70.812,-124.059,-25.891,28.549,-38.248
C03133=1013.526,70.570,-124.038,-25.878,28.484,-38.280
C03134=1013.530,70.330,-124.017,-25.866,28.418,-38.313
C03135=1013.533,70.089,-123.996,-25.853,28.354,-38.346
C03136=1013.536,69.848,-123.974,-25.841,28.289,-38.379
C03137=1013.538,69.607,-123.954,-25.828,28.225,-38.412
C03138=1013.541,69.366,-123.933,-25.815,28.160,-38.445
C03139=1013.544,69.123,-123.910,-25.803,28.096,-38.478
C03140=1013.547,68.878,-123.889,-25.790,28.030,-38.511
C03141=1013.550,68.629,-123.867,-25.777,27.964,-38.545
C03142=1013.553,68.380,-123.845,-25.764,27.899,-38.579
C03143=1013.556,68.131,-123.824,-25.751,27.834,-38.612
C03144=1013.559,67.885,-123.802,-25.738,27.769,-38.645
C03145=1013.562,67.644,-123.781,-25.725,27.706,-38.679
C03146=1013.564,67.406,-123.759,-25.713,27.645,-38.711
C03147=1013.567,67.168,-123.739,-25.700,27.583,-38.744
C03148=1013.570,66.932,-123.719,-25.688,27.522,-38.775
C03149=1013.572,66.695,-123.697,-25.676,27.461,-38.807
C03150=1013.575,66.460,-123.677,-25.663,27.400,-38.839
C03151=1013.580,66.057,-123.642,-25.642,27.298,-38.893
C03152=1013.582,65.854,-123.623,-25.632,27.247,-38.921
C03153=1013.584,65.622,-123.603,-25.619,27.187,-38.952
C03154=1013.588,65.379,-123.582,-25.607,27.126,-38.985
C03155=1013.591,65.126,-123.560,-25.593,27.062,-39.019
C03156=1013.593,64.866,-123.536,-25.580,26.997,-39.054
C03157=1013.596,64.600,-123.513,-25.566,26.931,-39.089
C03158=1013.599,64.331,-123.489,-25.552,26.865,-39.125
C03159=1013.602,64.063,-123.466,-25.538,26.798,-39.161
C03160=1013.605,63.810,-123.444,-25.525,26.736,-39.194
C03161=1013.607,63.572,-123.423,-25.513,26.677,-39.227
C03162=1013.611,63.322,-123.401,-25.500,26.616,-39.259
C03163=1013.613,63.039,-123.376,-25.485,26.547,-39.297
C03164=1013.616,62.744,-123.350,-25.470,26.475,-39.336
C03165=1013.620,62.469,-123.326,-25.455,26.409,-39.372
C03166=1013.623,62.182,-123.301,-25.440,26.339,-39.411
C03167=1013.626,61.905,-123.276,-25.426,26.274,-39.447
C03168=1013.628,61.669,-123.256,-25.414,26.217,-39.478
C03169=1013.631,61.433,-123.235,-25.402,26.161,-39.510
C03170=1013.634,61.199,-123.214,-25.389,26.105,-39.541
C03171=1013.636,60.963,-123.193,-25.377,26.050,-39.572
C03172=1013.639,60.727,-123.172,-25.365,25.994,-39.604
C03173=1013.641,60.491,-123.152,-25.353,25.939,-39.633
C03174=1013.644,60.257,-123.131,-25.340,25.884,-39.665
C03175=1013.646,60.021,-123.111,-25.328,25.829,-39.695
C03176=1013.649,59.785,-123.090,-25.316,25.775,-39.726
C03177=1013.652,59.549,-123.069,-25.304,25.719,-39.757
C03178=1013.654,59.313,-123.049,-25.292,25.665,-39.788
C03179=1013.657,59.078,-123.027,-25.280,25.611,-39.819
C03180=1013.659,58.843,-123.007,-25.268,25.558,-39.850
C03181=1013.662,58.607,-122.986,-25.255,25.504,-39.880
C03182=1013.664,58.371,-122.966,-25.243,25.451,-39.910
C03183=1013.667,58.136,-122.944,-25.231,25.398,-39.941
C03184=1013.669,57.901,-122.924,-25.219,25.345,-39.972
C03185=1013.671,57.665,-122.903,-25.207,25.292,-40.002
C03186=1013.673,57.429,-122.883,-25.195,25.239,-40.033
C03187=1013.676,57.193,-122.861,-25.183,25.187,-40.063
C03188=1013.678,56.958,-122.841,-25.171,25.134,-40.093
C03189=1013.681,56.722,-122.821,-25.159,25.083,-40.123
C03190=1013.683,56.487,-122.800,-25.147,25.031,-40.153
C03191=1013.685,56.252,-122.779,-25.135,24.979,-40.183
C03192=1013.688,56.016,-122.758,-25.123,24.928,-40.214
C03193=1013.690,55.780,-122.738,-25.111,24.877,-40.244
C03194=1013.693,55.545,-122.717,-25.099,24.826,-40.273
C03195=1013.695,55.309,-122.696,-25.087,24.775,-40.304
C03196=1013.698,55.073,-122.676,-25.075,24.724,-40.333
C03197=1013.700,54.838,-122.655,-25.063,24.674,-40.364
C03198=1013.702,54.602,-122.635,-25.051,24.623,-40.393
C03199=1013.704,54.367,-122.613,-25.039,24.573,-40.422
C03200=1013.706,54.131,-122.593,-25.028,24.524,-40.452
C03201=1013.710,53.896,-122.572,-25.016,24.474,-40.482
C03202=1013.711,53.660,-122.551,-25.004,24.424,-40.511
C03203=1013.713,53.425,-122.531,-24.992,24.375,-40.541
C03204=1013.716,53.189,-122.510,-24.980,24.327,-40.570
C03205=1013.718,52.953,-122.490,-24.968,24.278,-40.600
C03206=1013.720,52.718,-122.469,-24.956,24.228,-40.630
C03207=1013.723,52.483,-122.448,-24.945,24.180,-40.658
C03208=1013.725,52.247,-122.428,-24.933,24.132,-40.687
C03209=1013.727,52.012,-122.407,-24.921,24.084,-40.716
C03210=1013.730,51.776,-122.386,-24.910,24.037,-40.745
C03211=1013.732,51.540,-122.366,-24.898,23.989,-40.776
C03212=1013.733,51.305,-122.345,-24.886,23.942,-40.804
C03213=1013.736,51.069,-122.324,-24.875,23.894,-40.833
C03214=1013.738,50.833,-122.304,-24.863,23.847,-40.862
C03215=1013.741,50.599,-122.283,-24.851,23.800,-40.891
C03216=1013.743,50.363,-122.262,-24.840,23.754,-40.920
C03217=1013.745,50.127,-122.242,-24.828,23.708,-40.948
C03218=1013.747,49.892,-122.221,-24.816,23.662,-40.977
C03219=1013.749,49.656,-122.200,-24.805,23.615,-41.006
C03220=1013.752,49.420,-122.180,-24.793,23.570,-41.034
C03221=1013.754,49.185,-122.158,-24.782,23.524,-41.062
C03222=1013.756,48.950,-122.139,-24.770,23.478,-41.091
C03223=1013.758,48.715,-122.118,-24.759,23.433,-41.119
C03224=1013.760,48.479,-122.097,-24.748,23.388,-41.147
C03225=1013.763,48.243,-122.076,-24.736,23.344,-41.176
C03226=1013.765,48.008,-122.056,-24.725,23.299,-41.204
C03227=1013.766,47.773,-122.035,-24.713,23.254,-41.232
C03228=1013.768,47.537,-122.015,-24.702,23.211,-41.259
C03229=1013.770,47.302,-121.994,-24.691,23.166,-41.289
C03230=1013.773,47.067,-121.974,-24.679,23.123,-41.316
C03231=1013.776,46.831,-121.953,-24.668,23.079,-41.344
C03232=1013.777,46.596,-121.932,-24.657,23.035,-41.372
C03233=1013.779,46.360,-121.911,-24.646,22.992,-41.398
C03234=1013.781,46.124,-121.891,-24.634,22.950,-41.426
C03235=1013.783,45.889,-121.870,-24.623,22.906,-41.454
C03236=1013.785,45.654,-121.850,-24.612,22.864,-41.481
C03237=1013.787,45.418,-121.829,-24.601,22.821,-41.510
C03238=1013.789,45.183,-121.809,-24.590,22.779,-41.536
C03239=1013.791,44.948,-121.788,-24.579,22.737,-41.563
C03240=1013.793,44.713,-121.768,-24.568,22.695,-41.590
C03241=1013.795,44.477,-121.747,-24.557,22.654,-41.617
C03242=1013.798,44.242,-121.726,-24.546,22.612,-41.645
C03243=1013.800,44.006,-121.705,-24.534,22.571,-41.672
C03244=1013.801,43.771,-121.684,-24.523,22.530,-41.699
C03245=1013.803,43.535,-121.664,-24.513,22.489,-41.725
C03246=1013.805,43.300,-121.643,-24.502,22.448,-41.753
C03247=1013.808,43.065,-121.623,-24.491,22.408,-41.779
C03248=1013.810,42.829,-121.603,-24.480,22.369,-41.805
C03249=1013.811,42.594,-121.582,-24.469,22.328,-41.833
C03250=1013.814,42.358,-121.561,-24.458,22.288,-41.859
C03251=1013.814,42.124,-121.541,-24.447,22.248,-41.885
C03252=1013.817,41.888,-121.521,-24.437,22.209,-41.911
C03253=1013.818,41.653,-121.500,-24.426,22.170,-41.937
C03254=1013.820,41.417,-121.479,-24.415,22.131,-41.964
C03255=1013.822,41.182,-121.458,-24.405,22.092,-41.989
C03256=1013.825,40.947,-121.438,-24.394,22.053,-42.016
C03257=1013.826,40.712,-121.417,-24.384,22.015,-42.041
C03258=1013.828,40.476,-121.397,-24.373,21.976,-42.067
C03259=1013.830,40.241,-121.376,-24.362,21.938,-42.094
C03260=1013.832,40.006,-121.356,-24.352,21.900,-42.119
C03261=1013.834,39.770,-121.335,-24.341,21.863,-42.145
C03262=1013.835,39.535,-121.315,-24.331,21.826,-42.169
C03263=1013.837,39.300,-121.294,-24.320,21.788,-42.195
C03264=1013.839,39.064,-121.274,-24.310,21.751,-42.221
C03265=1013.841,38.829,-121.253,-24.300,21.714,-42.246
C03266=1013.843,38.594,-121.233,-24.289,21.677,-42.272
C03267=1013.845,38.359,-121.212,-24.279,21.641,-42.296
C03268=1013.852,37.261,-121.116,-24.235,21.484,-42.405
C03269=1013.855,36.913,-121.086,-24.234,21.485,-42.409
C03270=1013.858,36.514,-121.051,-24.233,21.484,-42.414
C03271=1013.861,36.114,-121.016,-24.233,21.485,-42.418
C03272=1013.864,35.714,-120.982,-24.232,21.486,-42.424
C03273=1013.867,35.314,-120.947,-24.231,21.486,-42.428
C03274=1013.869,34.914,-120.912,-24.231,21.486,-42.433
C03275=1013.872,34.515,-120.877,-24.230,21.486,-42.437
C03276=1013.875,34.115,-120.842,-24.229,21.487,-42.442
C03277=1013.878,33.716,-120.808,-24.229,21.488,-42.446
C03278=1013.881,33.316,-120.773,-24.228,21.487,-42.451
C03279=1013.884,32.917,-120.738,-24.228,21.489,-42.455
C03280=1013.886,32.517,-120.703,-24.227,21.489,-42.461
C03281=1013.888,32.117,-120.669,-24.226,21.489,-42.464
C03282=1013.892,31.717,-120.634,-24.226,21.489,-42.469
C03283=1013.894,31.318,-120.599,-24.225,21.490,-42.474
C03284=1013.897,30.918,-120.564,-24.224,21.490,-42.479
C03285=1013.899,30.518,-120.530,-24.224,21.491,-42.483
C03286=1013.902,30.120,-120.495,-24.223,21.491,-42.488
C03287=1013.905,29.719,-120.460,-24.223,21.492,-42.492
C03288=1013.907,29.320,-120.426,-24.222,21.492,-42.497
C03289=1013.909,28.921,-120.391,-24.221,21.492,-42.501
C03290=1013.912,28.522,-120.357,-24.221,21.493,-42.507
C03291=1013.915,28.122,-120.322,-24.220,21.493,-42.510
C03292=1013.916,27.722,-120.287,-24.219,21.493,-42.516
C03293=1013.919,27.323,-120.253,-24.219,21.495,-42.520
C03294=1013.921,26.924,-120.218,-24.218,21.494,-42.525
C03295=1013.923,26.525,-120.184,-24.218,21.495,-42.529
C03296=1013.925,26.125,-120.150,-24.217,21.496,-42.534
C03297=1013.928,25.726,-120.115,-24.216,21.496,-42.540
C03298=1013.930,25.326,-120.080,-24.215,21.496,-42.543
C03299=1013.932,24.928,-120.046,-24.215,21.497,-42.549
C03300=1013.934,24.528,-120.012,-24.214,21.497,-42.553
C03301=1013.937,24.129,-119.977,-24.213,21.497,-42.558
C03302=1013.939,23.745,-119.944,-24.213,21.498,-42.562
C03303=1013.941,23.416,-119.916,-24.213,21.498,-42.564
C03304=1013.942,23.144,-119.892,-24.212,21.498,-42.567
C03305=1013.943,22.909,-119.872,-24.211,21.499,-42.573
C03306=1013.944,22.677,-119.852,-24.211,21.500,-42.577
C03307=1013.947,22.411,-119.829,-24.211,21.500,-42.580
C03308=1013.947,22.089,-119.801,-24.210,21.500,-42.584
C03309=1013.950,21.715,-119.769,-24.210,21.501,-42.586
C03310=1013.951,21.300,-119.733,-24.209,21.501,-42.593
C03311=1013.952,21.056,-119.711,-24.208,21.501,-42.597
C03312=1013.954,20.784,-119.689,-24.208,21.502,-42.599
C03313=1013.955,20.493,-119.663,-24.207,21.501,-42.602
C03314=1013.956,20.196,-119.638,-24.207,21.501,-42.604
C03315=1013.958,19.909,-119.614,-24.207,21.503,-42.606
C03316=1013.959,19.643,-119.590,-24.206,21.502,-42.610
C03317=1013.960,19.407,-119.570,-24.206,21.503,-42.613
C03318=1013.963,18.997,-119.535,-24.205,21.503,-42.619
C03319=1013.963,18.799,-119.518,-24.205,21.503,-42.622
C03320=1013.965,18.402,-119.483,-24.204,21.503,-42.626
C03321=1013.967,18.007,-119.450,-24.203,21.504,-42.632
C03322=1013.968,17.612,-119.416,-24.203,21.505,-42.635
C03323=1013.970,17.218,-119.383,-24.202,21.505,-42.641
C03324=1013.972,16.824,-119.348,-24.201,21.505,-42.646
C03325=1013.973,16.431,-119.315,-24.201,21.506,-42.650
C03326=1013.975,16.039,-119.281,-24.200,21.506,-42.656
C03327=1013.977,15.649,-119.248,-24.200,21.507,-42.659
C03328=1013.979,15.259,-119.214,-24.199,21.507,-42.665
C03329=1013.980,14.869,-119.180,-24.198,21.508,-42.670
C03330=1013.981,14.480,-119.148,-24.198,21.508,-42.674
C03331=1013.983,14.092,-119.114,-24.197,21.509,-42.680
C03332=1013.984,13.704,-119.081,-24.196,21.509,-42.683
C03333=1013.986,13.317,-119.048,-24.196,21.509,-42.689
C03334=1013.987,12.931,-119.015,-24.195,21.511,-42.693
C03335=1013.989,12.543,-118.982,-24.194,21.510,-42.698
C03336=1013.990,12.157,-118.949,-24.193,21.510,-42.703
C03337=1013.992,11.771,-118.916,-24.193,21.512,-42.707
C03338=1013.993,11.384,-118.882,-24.192,21.511,-42.713
C03339=1013.994,10.999,-118.850,-24.192,21.512,-42.716
C03340=1013.995,10.616,-118.818,-24.191,21.513,-42.722
C03341=1013.997,10.235,-118.785,-24.191,21.513,-42.726
C03342=1013.997,9.857,-118.752,-24.190,21.513,-42.731
C03343=1013.999,9.480,-118.720,-24.189,21.514,-42.737
C03344=1014.000,9.105,-118.689,-24.189,21.514,-42.740
C03345=1014.001,8.728,-118.657,-24.188,21.515,-42.746
C03346=1014.003,8.351,-118.624,-24.187,21.515,-42.751
C03347=1014.003,7.969,-118.591,-24.187,21.516,-42.755
C03348=1014.004,7.586,-118.559,-24.186,21.516,-42.761
C03349=1014.005,7.198,-118.526,-24.185,21.517,-42.764
C03350=1014.007,6.807,-118.493,-24.185,21.517,-42.770
C03351=1014.007,6.415,-118.460,-24.184,21.517,-42.775
C03352=1014.009,6.022,-118.427,-24.183,21.519,-42.779
C03353=1014.010,5.628,-118.393,-24.182,21.518,-42.785
C03354=1014.010,5.234,-118.359,-24.182,21.519,-42.790
C03355=1014.012,4.839,-118.326,-24.181,21.520,-42.794
C03356=1014.012,4.443,-118.293,-24.180,21.519,-42.799
C03357=1014.014,4.048,-118.258,-24.180,21.520,-42.805
C03358=1014.014,3.658,-118.225,-24.179,21.521,-42.809
C03359=1014.015,3.299,-118.195,-24.179,21.521,-42.812
C03360=1014.016,2.971,-118.167,-24.178,21.521,-42.817
C03361=1014.016,2.657,-118.141,-24.177,21.522,-42.823
C03362=1014.017,2.335,-118.114,-24.177,21.522,-42.827
C03363=1014.017,1.982,-118.083,-24.176,21.523,-42.833
C03364=1014.018,1.596,-118.051,-24.175,21.524,-42.836
C03365=1014.019,1.199,-118.017,-24.175,21.523,-42.841
C03366=1014.020,0.799,-117.984,-24.174,21.525,-42.846
C03367=1014.021,0.400,-117.951,-24.173,21.525,-42.851
C03368=1014.022,-0.002,-117.917,-24.173,21.525,-42.857
C03369=1014.022,-0.406,-117.882,-24.172,21.525,-42.862
C03370=1014.023,-0.811,-117.848,-24.171,21.526,-42.867
C03371=1014.023,-1.219,-117.813,-24.171,21.527,-42.872
C03372=1014.024,-1.629,-117.779,-24.170,21.527,-42.877
C03373=1014.025,-2.041,-117.744,-24.169,21.528,-42.882
C03374=1014.025,-2.457,-117.709,-24.169,21.529,-42.888
C03375=1014.026,-2.874,-117.674,-24.168,21.529,-42.893
C03376=1014.026,-3.293,-117.639,-24.167,21.529,-42.899
C03377=1014.027,-3.714,-117.604,-24.166,21.530,-42.904
C03378=1014.026,-3.926,-117.586,-24.166,21.530,-42.908
C03379=1014.026,-4.138,-117.567,-24.165,21.530,-42.910
C03380=1014.027,-4.352,-117.550,-24.165,21.530,-42.913
C03381=1014.027,-4.567,-117.532,-24.165,21.531,-42.915
C03382=1014.027,-4.784,-117.513,-24.164,21.531,-42.919
C03383=1014.028,-5.003,-117.495,-24.164,21.531,-42.921
C03384=1014.028,-5.222,-117.477,-24.163,21.532,-42.925
C03385=1014.028,-5.443,-117.458,-24.163,21.532,-42.927
C03386=1014.029,-5.666,-117.440,-24.163,21.532,-42.930
C03387=1014.029,-5.890,-117.421,-24.162,21.532,-42.934
C03388=1014.029,-6.113,-117.402,-24.162,21.533,-42.935
C03389=1014.029,-6.338,-117.383,-24.161,21.533,-42.939
C03390=1014.029,-6.562,-117.365,-24.161,21.533,-42.941
C03391=1014.029,-6.787,-117.346,-24.161,21.533,-42.944
C03392=1014.029,-7.009,-117.327,-24.160,21.534,-42.947
C03393=1014.029,-7.232,-117.309,-24.160,21.534,-42.950
C03394=1014.029,-7.453,-117.289,-24.160,21.535,-42.952
C03395=1014.030,-7.673,-117.271,-24.159,21.534,-42.956
C03396=1014.030,-7.893,-117.253,-24.159,21.535,-42.959
C03397=1014.030,-8.111,-117.235,-24.158,21.535,-42.961
C03398=1014.030,-8.328,-117.217,-24.158,21.536,-42.965
C03399=1014.030,-8.545,-117.198,-24.158,21.536,-42.967
C03400=1014.030,-8.762,-117.180,-24.157,21.536,-42.971
C03401=1014.030,-8.979,-117.162,-24.157,21.537,-42.973
C03402=1014.030,-9.195,-117.144,-24.156,21.536,-42.976
C03403=1014.030,-9.411,-117.126,-24.156,21.537,-42.980
C03404=1014.030,-9.628,-117.107,-24.156,21.537,-42.982
C03405=1014.031,-9.844,-117.090,-24.155,21.538,-42.985
C03406=1014.030,-10.060,-117.071,-24.155,21.538,-42.987
C03407=1014.030,-10.276,-117.054,-24.154,21.538,-42.991
C03408=1014.030,-10.491,-117.035,-24.154,21.539,-42.993
C03409=1014.030,-10.707,-117.018,-24.154,21.538,-42.996
C03410=1014.030,-10.922,-117.000,-24.153,21.539,-42.998
C03411=1014.030,-11.137,-116.981,-24.153,21.539,-43.002
C03412=1014.030,-11.351,-116.964,-24.152,21.539,-43.006
C03413=1014.029,-11.565,-116.946,-24.152,21.540,-43.007
C03414=1014.030,-11.778,-116.929,-24.152,21.540,-43.011
C03415=1014.030,-11.991,-116.910,-24.151,21.540,-43.013
C03416=1014.029,-12.203,-116.893,-24.151,21.540,-43.016
C03417=1014.030,-12.415,-116.875,-24.151,21.541,-43.019
C03418=1014.030,-12.626,-116.857,-24.150,21.541,-43.022
C03419=1014.030,-13.047,-116.822,-24.149,21.542,-43.028
C03420=1014.029,-13.257,-116.805,-24.149,21.542,-43.029
C03421=1014.029,-13.674,-116.770,-24.148,21.543,-43.035
C03422=1014.029,-14.089,-116.736,-24.148,21.543,-43.041
C03423=1014.029,-14.500,-116.701,-24.147,21.544,-43.046
C03424=1014.029,-14.909,-116.667,-24.146,21.544,-43.052
C03425=1014.028,-15.314,-116.634,-24.145,21.545,-43.057
C03426=1014.028,-15.717,-116.600,-24.145,21.545,-43.063
C03427=1014.027,-16.118,-116.567,-24.144,21.546,-43.068
C03428=1014.027,-16.518,-116.534,-24.143,21.546,-43.074
C03429=1014.026,-16.916,-116.501,-24.142,21.547,-43.079
C03430=1014.026,-17.314,-116.468,-24.142,21.548,-43.085
C03431=1014.026,-17.712,-116.435,-24.141,21.547,-43.090
C03432=1014.025,-18.123,-116.401,-24.140,21.548,-43.098
C03433=1014.025,-18.371,-116.380,-24.139,21.549,-43.101
C03434=1014.025,-18.658,-116.356,-24.139,21.549,-43.105
C03435=1014.024,-18.970,-116.331,-24.139,21.550,-43.107
C03436=1014.023,-19.281,-116.305,-24.139,21.550,-43.109
C03437=1014.023,-19.570,-116.281,-24.138,21.550,-43.113
C03438=1014.023,-19.819,-116.260,-24.138,21.551,-43.116
C03439=1014.022,-20.230,-116.227,-24.136,21.551,-43.123
C03440=1014.021,-20.627,-116.193,-24.136,21.552,-43.129
C03441=1014.021,-21.025,-116.161,-24.135,21.553,-43.135
C03442=1014.020,-21.423,-116.128,-24.134,21.552,-43.140
C03443=1014.020,-21.820,-116.095,-24.134,21.553,-43.146
C03444=1014.018,-22.218,-116.062,-24.133,21.554,-43.151
C03445=1014.018,-22.615,-116.029,-24.132,21.554,-43.156
C03446=1014.017,-23.013,-115.997,-24.131,21.555,-43.162
C03447=1014.016,-23.410,-115.964,-24.131,21.555,-43.168
C03448=1014.016,-23.807,-115.931,-24.130,21.556,-43.173
C03449=1014.014,-24.205,-115.898,-24.129,21.556,-43.178
C03450=1014.014,-24.602,-115.866,-24.128,21.557,-43.184
C03451=1014.013,-25.001,-115.833,-24.128,21.558,-43.190
C03452=1014.012,-25.397,-115.800,-24.127,21.558,-43.195
C03453=1014.011,-25.795,-115.768,-24.126,21.558,-43.201
C03454=1014.010,-26.193,-115.735,-24.125,21.559,-43.206
C03455=1014.008,-26.591,-115.703,-24.125,21.560,-43.212
C03456=1014.007,-26.988,-115.670,-24.124,21.560,-43.217
C03457=1014.006,-27.385,-115.637,-24.123,21.561,-43.221
C03458=1014.005,-27.783,-115.605,-24.123,21.562,-43.227
C03459=1014.005,-28.181,-115.572,-24.122,21.562,-43.232
C03460=1014.003,-28.578,-115.539,-24.121,21.562,-43.238
C03461=1014.001,-28.975,-115.507,-24.120,21.563,-43.243
C03462=1014.000,-29.373,-115.475,-24.120,21.564,-43.249
C03463=1013.999,-29.771,-115.442,-24.119,21.565,-43.255
C03464=1013.998,-30.167,-115.409,-24.118,21.565,-43.260
C03465=1013.996,-30.565,-115.377,-24.117,21.565,-43.265
C03466=1013.995,-30.963,-115.344,-24.117,21.566,-43.271
C03467=1013.994,-31.361,-115.312,-24.116,21.567,-43.277
C03468=1013.992,-31.758,-115.279,-24.115,21.568,-43.282
C03469=1013.990,-32.155,-115.247,-24.114,21.567,-43.287
C03470=1013.989,-32.553,-115.215,-24.114,21.568,-43.293
C03471=1013.987,-32.950,-115.183,-24.113,21.569,-43.299
C03472=1013.986,-33.348,-115.149,-24.112,21.570,-43.304
C03473=1013.985,-33.745,-115.117,-24.111,21.570,-43.310
C03474=1013.983,-34.143,-115.085,-24.111,21.570,-43.315
C03475=1013.981,-34.540,-115.052,-24.110,21.571,-43.321
C03476=1013.980,-34.937,-115.020,-24.109,21.571,-43.328
C03477=1013.978,-35.335,-114.988,-24.108,21.572,-43.334
C03478=1013.976,-35.732,-114.956,-24.107,21.572,-43.339
C03479=1013.974,-36.130,-114.923,-24.107,21.573,-43.344
C03480=1013.972,-36.527,-114.891,-24.106,21.573,-43.350
C03481=1013.971,-36.924,-114.859,-24.105,21.574,-43.356
C03482=1013.969,-37.322,-114.826,-24.105,21.575,-43.361
C03483=1013.967,-37.719,-114.794,-24.104,21.575,-43.366
C03484=1013.965,-38.117,-114.762,-24.103,21.576,-43.372
C03485=1013.963,-38.515,-114.730,-24.102,21.576,-43.378
C03486=1013.961,-38.911,-114.698,-24.102,21.577,-43.383
C03487=1013.960,-39.309,-114.665,-24.101,21.578,-43.389
C03488=1013.958,-39.706,-114.633,-24.100,21.578,-43.394
C03489=1013.955,-40.103,-114.600,-24.099,21.579,-43.400
C03490=1013.953,-40.501,-114.568,-24.099,21.579,-43.405
C03491=1013.951,-40.899,-114.536,-24.098,21.580,-43.411
C03492=1013.949,-41.296,-114.504,-24.097,21.581,-43.417
C03493=1013.947,-41.693,-114.472,-24.096,21.582,-43.422
C03494=1013.945,-42.090,-114.440,-24.096,21.582,-43.427
C03495=1013.942,-42.487,-114.408,-24.095,21.582,-43.433
C03496=1013.940,-42.885,-114.376,-24.094,21.583,-43.439
C03497=1013.937,-43.282,-114.344,-24.093,21.584,-43.444
C03498=1013.935,-43.679,-114.312,-24.092,21.584,-43.451
C03499=1013.933,-44.077,-114.280,-24.092,21.585,-43.457
C03500=1013.931,-44.474,-114.247,-24.091,21.585,-43.462
C03501=1013.928,-44.871,-114.216,-24.090,21.585,-43.468
C03502=1013.926,-45.269,-114.184,-24.089,21.586,-43.473
C03503=1013.922,-45.666,-114.152,-24.089,21.587,-43.479
C03504=1013.915,-46.816,-114.059,-24.139,21.774,-43.378
C03505=1013.914,-47.049,-114.040,-24.150,21.815,-43.356
C03506=1013.912,-47.283,-114.021,-24.162,21.858,-43.333
C03507=1013.911,-47.516,-114.002,-24.173,21.901,-43.310
C03508=1013.909,-47.751,-113.984,-24.185,21.943,-43.287
C03509=1013.907,-47.985,-113.965,-24.196,21.986,-43.264
C03510=1013.906,-48.218,-113.946,-24.208,22.031,-43.240
C03511=1013.905,-48.452,-113.927,-24.220,22.074,-43.215
C03512=1013.903,-48.686,-113.908,-24.232,22.118,-43.192
C03513=1013.901,-48.920,-113.890,-24.243,22.162,-43.168
C03514=1013.899,-49.153,-113.871,-24.255,22.207,-43.144
C03515=1013.898,-49.387,-113.852,-24.267,22.253,-43.120
C03516=1013.897,-49.620,-113.833,-24.279,22.297,-43.096
C03517=1013.894,-49.854,-113.814,-24.291,22.343,-43.071
C03518=1013.893,-50.088,-113.796,-24.303,22.388,-43.047
C03519=1013.891,-50.322,-113.777,-24.315,22.434,-43.022
C03520=1013.890,-50.555,-113.758,-24.328,22.480,-42.997
C03521=1013.887,-50.789,-113.739,-24.340,22.528,-42.972
C03522=1013.886,-51.023,-113.721,-24.352,22.574,-42.947
C03523=1013.885,-51.257,-113.702,-24.364,22.621,-42.922
C03524=1013.882,-51.490,-113.683,-24.377,22.669,-42.897
C03525=1013.881,-51.724,-113.664,-24.389,22.716,-42.871
C03526=1013.879,-51.958,-113.646,-24.402,22.765,-42.846
C03527=1013.877,-52.191,-113.627,-24.414,22.813,-42.820
C03528=1013.876,-52.425,-113.608,-24.427,22.862,-42.793
C03529=1013.873,-52.659,-113.590,-24.440,22.910,-42.768
C03530=1013.872,-52.892,-113.570,-24.453,22.960,-42.741
C03531=1013.870,-53.126,-113.552,-24.465,23.009,-42.715
C03532=1013.869,-53.359,-113.534,-24.478,23.059,-42.689
C03533=1013.866,-53.593,-113.514,-24.491,23.109,-42.663
C03534=1013.864,-53.827,-113.496,-24.504,23.159,-42.636
C03535=1013.863,-54.061,-113.477,-24.517,23.210,-42.609
C03536=1013.861,-54.293,-113.458,-24.530,23.261,-42.583
C03537=1013.859,-54.528,-113.439,-24.543,23.312,-42.556
C03538=1013.857,-54.761,-113.421,-24.556,23.364,-42.529
C03539=1013.856,-54.995,-113.402,-24.569,23.415,-42.502
C03540=1013.854,-55.228,-113.384,-24.582,23.467,-42.475
C03541=1013.851,-55.462,-113.364,-24.596,23.520,-42.446
C03542=1013.849,-55.696,-113.346,-24.609,23.572,-42.418
C03543=1013.848,-55.930,-113.327,-24.622,23.625,-42.392
C03544=1013.845,-56.163,-113.308,-24.636,23.679,-42.364
C03545=1013.844,-56.397,-113.290,-24.649,23.732,-42.336
C03546=1013.841,-56.631,-113.271,-24.663,23.786,-42.307
C03547=1013.840,-56.866,-113.252,-24.676,23.841,-42.280
C03548=1013.838,-57.099,-113.234,-24.690,23.895,-42.251
C03549=1013.836,-57.334,-113.215,-24.704,23.950,-42.222
C03550=1013.834,-57.568,-113.196,-24.717,24.005,-42.194
C03551=1013.831,-57.802,-113.178,-24.731,24.061,-42.165
C03552=1013.830,-58.037,-113.159,-24.745,24.116,-42.137
C03553=1013.828,-58.271,-113.140,-24.759,24.173,-42.107
C03554=1013.825,-58.507,-113.120,-24.773,24.230,-42.078
C03555=1013.824,-58.742,-113.102,-24.787,24.287,-42.049
C03556=1013.822,-58.978,-113.084,-24.801,24.344,-42.020
C03557=1013.819,-59.213,-113.064,-24.815,24.401,-41.990
C03558=1013.817,-59.449,-113.045,-24.828,24.459,-41.961
C03559=1013.815,-59.685,-113.027,-24.843,24.518,-41.932
C03560=1013.813,-59.921,-113.008,-24.857,24.577,-41.901
C03561=1013.811,-60.156,-112.989,-24.871,24.636,-41.872
C03562=1013.808,-60.393,-112.970,-24.886,24.695,-41.842
C03563=1013.806,-60.631,-112.952,-24.900,24.756,-41.811
C03564=1013.804,-60.866,-112.933,-24.915,24.816,-41.780
C03565=1013.802,-61.103,-112.913,-24.929,24.877,-41.749
C03566=1013.799,-61.341,-112.895,-24.944,24.938,-41.719
C03567=1013.797,-61.579,-112.876,-24.958,24.999,-41.688
C03568=1013.796,-61.816,-112.857,-24.973,25.060,-41.658
C03569=1013.793,-62.054,-112.838,-24.988,25.122,-41.626
C03570=1013.791,-62.292,-112.819,-25.002,25.184,-41.595
C03571=1013.789,-62.530,-112.800,-25.017,25.247,-41.563
C03572=1013.787,-62.768,-112.781,-25.032,25.310,-41.533
C03573=1013.784,-63.006,-112.761,-25.047,25.374,-41.500
C03574=1013.782,-63.245,-112.743,-25.062,25.437,-41.469
C03575=1013.779,-63.484,-112.723,-25.077,25.502,-41.437
C03576=1013.777,-63.723,-112.705,-25.092,25.566,-41.405
C03577=1013.775,-63.962,-112.685,-25.107,25.631,-41.373
C03578=1013.773,-64.201,-112.666,-25.122,25.697,-41.340
C03579=1013.770,-64.441,-112.647,-25.137,25.762,-41.309
C03580=1013.767,-64.679,-112.628,-25.152,25.828,-41.276
C03581=1013.765,-64.919,-112.609,-25.168,25.894,-41.243
